(* check controller parameters: (MinOutput > MaxOutput) *)
IF ( MinOutput > MaxOutput ) 
THEN
	ErrorID 												:= ERR_INVALIDPARAM;
	Error													:= TRUE;
	RETURN;
END_IF;

(* check inner and outer window parameters: outer window must be greater than the inner window *)
IF((bIsIPart) AND ( OuterWindow > 0.0 )) 
THEN
	IF (InnerWindow > OuterWindow) 
	THEN
		ErrorId 											:= ERR_INVALIDPARAM;
		Error												:= TRUE;
		RETURN;
	END_IF;
	bIsOuterWnd 											:= TRUE;
END_IF;

(* set internal init flag *)
bIsInitDone													:= TRUE;
Q		 													:= MinOutput;
reset													:= TRUE;
END_METHOD

METHOD PUBLIC synchronize : BOOL  //Return value = TRUE if execution finished
VAR_INPUT 
	IN											:	LREAL;
END_VAR
	MemSyncValue										:= IN;
	
	(* Demand:  SyncValue != Ysum  with  SyncValue = Ysum = YP + YI + YD  =>  YI = SyncValue - Yp - Yd *)
	IF 	( bIsIPart = TRUE ) 
	THEN	(* I-part exists independent from the D-part *)
		(* Normal:  fYI = fYI_1 + fDi * (fE + fE_1) *)
		fYD 											:= fYD_1	:= 0.0;								
		fYI												:= fYI_1	:= MemSyncValue - fYP - fYD;	
		fY												:= MemSyncValue;
	ELSIF ( bIsDPart = TRUE ) 
	THEN	(* no I-part available, only D-part exits *)
		(* Normal:  fYD = fCd * fYD_1 + fDd * (fE - fE_1) *)
		(* fYD := fYD_1 := (fSyncValue - fYP - fYI) / fCd;*)(* 1) pre-calculation for the next cycle; fYI must be zero because there exists no I-part *)
		fYD												:= fYD_1	:= (MemSyncValue - fYP - fYI);		(* 2) fYI must be zero because there exists no I-part *)
		fY												:= MemSyncValue;
	END_IF                              				
	
	Synchronize											:= TRUE;
END_METHOD

END_FUNCTION_BLOCK

// POUs/ControllerTools/PT1Filter
//Low pass filter with a programmable time Tn and factor Kp.
FUNCTION_BLOCK PT1Filter
VAR_INPUT
	Enable													:	BOOL ; 	// FB will be processed as long as enable is TRUE 
	In														:	LREAL := 0.0;	// Actual value
	ResetTrig												:	BOOL ; 	// The function block will be reset with a rising edge 
	Sync													:	BOOL ; 	// Synchronise In to Q - equivalent to Synchronize method
	Kp														:	LREAL := 1.0; 	// Gain
	Tn														:	TIME := T#1S; 	// Integral time 
	Cycletime 												:	TIME := T#10MS;	// cycletime 
END_VAR	            										
VAR_OUTPUT          										
	Q														: LREAL;			// Output
	Error													: BOOL;				// Rising edge of Error informs that an error occurred during the execution of the Function Block 
END_VAR             										
VAR                 	
	Q_old													: LREAL;
END_VAR

(**************************************************************************************
	formula: 
	y(k) = [1-T/T1]	* y(k-1)
			+ T/T1		* v 		* e(k) 
*************************************************************************************)

	Error 													:= Cycletime = T#0MS OR  tn = T#0MS OR Kp = 0.0;
                            								
	IF Enable               								
		AND NOT Error       								
	THEN                    								
		Q 													:=  (1- TIME_TO_LREAL(Cycletime) / TIME_TO_LREAL(Tn))	* Q_old
															 	+ TIME_TO_LREAL(Cycletime) / TIME_TO_LREAL(Tn)	* Kp		* In;
		Q_Old 												:= Q;
	ELSE //Hold
		;
	END_IF

	IF ResetTrig
	THEN
		reset();
	ELSIF Sync
	THEN
		Synchronize(IN);
	END_IF

(************************************************************************************)

METHOD reset : BOOL //Return value = TRUE if execution finished
VAR_INPUT
END_VAR
Q := Q_old 				:= 0.0;
reset				:= TRUE;
END_METHOD

METHOD PUBLIC synchronize : BOOL //Return value = TRUE if execution finished
VAR_INPUT
	IN						:	LREAL;
END_VAR
Q 	:= Q_Old 	 := IN;
Synchronize		:= TRUE;
END_METHOD

END_FUNCTION_BLOCK

// POUs/ControllerTools/signum
//LREAL Signum function
FUNCTION signum : LREAL
VAR_INPUT
	IN		:	LREAL;
END_VAR
VAR
END_VAR

IF IN = 0.0
THEN
	SIGNUM		:= 0.0;
ELSIF IN > 0.0
THEN
	SIGNUM		:= 1.0;
ELSE
	SIGNUM	 	:= -1.0;
END_IF

END_FUNCTION

// POUs/ControllerTools/SlewRateLimitter
//LREAL Slew rate limitter with a timebased change rate
FUNCTION_BLOCK SlewRateLimitter
VAR_INPUT
	IN														: LREAL := 0.0;	 //Actual value
	Sync													: BOOL := FALSE; //Sync signal sets IN to Q	
	Cycletime												: LREAL := 0.001; //cycletime in ms
	Rate													: LREAL := 1.0;	 // changes per second
END_VAR                 									
VAR_OUTPUT              									
	Q														: LREAL := 0.0;   //Output
END_VAR                 									
VAR                     	
	x														: LREAL := 0.0;
END_VAR

//Based on MC_AxUtiSlewRateLimitter_BkPlcMc from TcPlcLibHydraulics , Author WOs
IF Cycletime <= 0.0001 OR Rate <= 0.0 OR Sync
THEN
	Q														:= IN;
ELSE                    									
	x														:= Cycletime * Rate;
	IF ABS(IN) > X OR ABS(Q > In)
	THEN //Start ramping only after In is greater than Rate and as long as Q is greater (if In jumps to zero)
		Q													:= Q + LIMIT(-x , IN - Q , x); 		
	ELSE
		Q													:= In;
	END_IF
END_IF

METHOD PUBLIC synchronize : BOOL //Return value = TRUE if execution finished
VAR_INPUT
	IN														:	LREAL;
END_VAR
Q 															:= IN;
Synchronize 												:= TRUE;
END_METHOD

END_FUNCTION_BLOCK

// POUs/ControllerTools/SlidingAverage
FUNCTION_BLOCK SlidingAverage 
VAR_OUTPUT CONSTANT 
	MIN_BUFFER												:	INT := 1;
	MAX_BUFFER												:	INT := PARAM.SLIDING_AVERAGE_MAX_ENTRYS;
END_VAR
VAR_INPUT
	In														: LREAL := 0.0;			//Actual value 
	ResetTrig												: BOOL := FALSE;		//Reset average buffer
	MaxNoOfValues											: DINT := PARAM.SLIDING_AVERAGE_MAX_ENTRYS;//Buffer limit if value is smaller than MAX_BUFFER
	SampleTime												: TIME := T#0MS;
END_VAR                 									
VAR_OUTPUT              									
	Q														: LREAL := 0.0;			//Average value
	Derivative												: LREAL := 0.0;			//
	ActIdx													: DINT := 1; 			//rotating count of buffer 
	Buffer													: ARRAY [MIN_BUFFER..MAX_BUFFER] OF LREAL;
END_VAR                 									
VAR           
	MinIdx													: DINT := MIN_BUFFER;   
	MaxIdx													: DINT := 0;       									
	Count													: DINT := 0; // limited count 
	pBuffer													: POINTER TO LREAL := 0;
	pIdx													: POINTER TO LREAL := 0;
	IdxOld													: DINT := 1;
	ftotal													: LREAL;
	fttotal													: LREAL;
	tonSampleTimer											: ton;
END_VAR


IF ResetTrig THEN reset(); RETURN; END_IF

pBuffer														:= ADR(Buffer);
MaxIdx														:= LIMIT(MIN_BUFFER, TO_INT(MaxNoOfValues), MAX_BUFFER);

IF(ActIdx>MaxIdx)
THEN
	ActIdx													:= MinIdx;
END_IF                      								
IF(ActIdx<MinIdx)           								
THEN                        								
	ActIdx													:= MaxIdx;
END_IF                      								
                            								
IF(ActIdx>MaxIdx)           								
THEN                        								
	Q														:= IN; (* Puffer-Indices sind unsinnig *)
ELSIF(pBuffer=0)            								
THEN                        								
	Q														:= IN; (* Puffer-Adresse ist unsinnig *)
ELSE            
	tonSampleTimer(IN := SampleTime > T#0MS, PT :=  SampleTime);
	IF NOT tonSampleTimer.IN OR tonSampleTimer.Q    
	THEN   			
		tonSampleTimer(IN := FALSE);	
		
		Count												:= MIN(Count, MaxIdx - MinIdx + 1);
		IdxOld												:= ActIdx - Count;
															
		IF(IdxOld<MinIdx)      								
		THEN                    							
			IdxOld											:= IdxOld + MaxIdx - MinIdx + 1;
		END_IF                  	                        
									                        
		IF(ActIdx=MinIdx)       	                        
		THEN                    	                        
			fttotal											:= 0.0;
		END_IF                  							
															
		IF(Count<1)            								
		THEN                    							
			ftotal := Derivative 							:= 0.0;	(* first cycle *)
		END_IF                  							
															
		pIdx												:= pBuffer + ((ActIdx - MinIdx) * SIZEOF(LREAL));
									                        
		IF(Count = (MaxIdx - MinIdx + 1))                   
		THEN                                                
			Derivative										:= (IN - pIdx^) / DINT_TO_LREAL(Count);
			ftotal											:= ftotal-pIdx^;		(* buffer is filled at least once *)
		END_IF                  							
		pIdx^												:=IN;
		fttotal												:=fttotal + IN;
		ftotal												:=ftotal + IN;
															
		ActIdx												:=ActIdx + 1;
									                        
		IF(ActIdx > MaxIdx)                                 
		THEN                                                
			(* swapping *)                                  
			ftotal											:= fttotal;
			ActIdx											:= MinIdx;
		END_IF                                              
		                                                    
		Count												:= MIN(Count + 1, MaxIdx - MinIdx + 1);
															
		Q													:=ftotal / DINT_TO_LREAL(Count);
	END_IF
END_IF

METHOD PUBLIC reset : BOOL //Return value = TRUE if execution finished
VAR_INPUT
END_VAR
Q															:=0.0;
Derivative													:=0.0;
ActIdx														:=MIN_BUFFER;	(* rotating count *)
Count														:=0;			(* limited count *)
                        									
                        									
IdxOld														:=1;
                        	
ftotal														:=0.0;
fttotal														:=0.0;
MEMSET(ADR(Buffer), 0 , SIZEOF(Buffer));
reset													:= TRUE;
END_METHOD

END_FUNCTION_BLOCK

// POUs/ControllerTools/SlidingAverageExt
//LREAL Sliding average with dynamic allocation of memory according MaxNoofValues 
{attribute 'enable_dynamic_creation'}
FUNCTION_BLOCK SlidingAverageExt 
VAR_INPUT
	In														: LREAL := 0.0;			//Actual value 
	ResetTrig												: BOOL ;		//Reset average buffer
	MaxNoOfValues											: DINT (0..10000) := 0;//Size of buffer (Array size) needs to get assigend in declaration
	SampleTime												: TIME := T#0MS;
END_VAR                 									
VAR_OUTPUT              									
	Q														: LREAL := 0.0;			//Average value
	Derivative												: LREAL := 0.0;			//
	ActIdx													: DINT := 1; 			//rotating count of buffer 
END_VAR                 									
VAR       
	MaxIdx													: DINT := 0;      
	MinIdx													: DINT := 1;        									
	Count													: DINT := 0; // limited count 
	pBuffer													: POINTER TO LREAL := 0;
	pIdx													: POINTER TO LREAL := 0;
	IdxOld													: DINT := 1;
	ftotal													: LREAL;
	fttotal													: LREAL;
	tonSampleTimer											: ton;
END_VAR

(* be sure to have nIdx inside MinIdx..MaxIdx *)
IF pBuffer = 0 AND MaxNoOfValues > 0
THEN //Alocate buffer memory
	pBuffer 												:= __NEW(LREAL,TO_UDINT(MaxNoOfValues)); 	
	IF NOT PARAM.ENABLE_DEBUG_MSG_DYNAMIC_MEM_ALLOCATION
	THEN 
		;
	ELSIF MaxIdx = 0 
	THEN
		AdsLogHint('EngineeringToolbox | FB SlidingAverageExt | An instance allocated %s bytes from the dynamic memory of the ADS router memory pool', TO_STRING(MaxNoOfValues * SIZEOF(LREAL)));	
	ELSE //Allocation of additional memory space
		AdsLogWarn('EngineeringToolbox | FB SlidingAverageExt | Value of "MaxNoOfValues" changed and one instance allocated additional %s bytes from the dynamic memory of the ADS router memory pool', TO_STRING(MaxNoOfValues * SIZEOF(LREAL)));
	END_IF
	MinIdx													:= 1;
	MaxIdx													:= MaxNoOfValues;
ELSIF MaxNoOfValues <> MaxIdx OR MaxNoOfValues = 0
THEN
	reset();
	FB_exit(FALSE);
	RETURN;
END_IF

IF ResetTrig THEN reset(); RETURN; END_IF

IF(ActIdx>MaxIdx)
THEN
	ActIdx													:= MinIdx;
END_IF                      								
IF(ActIdx<MinIdx)           								
THEN                        								
	ActIdx													:= MaxIdx;
END_IF                      								
                            								
IF(ActIdx>MaxIdx)           								
THEN                        								
	Q														:= IN; (* Puffer-Indices sind unsinnig *)
ELSIF(pBuffer=0)            								
THEN                        								
	Q														:= IN; (* Puffer-Adresse ist unsinnig *)
ELSE       
	tonSampleTimer(IN := SampleTime > T#0MS, PT :=  SampleTime);
	IF NOT tonSampleTimer.IN OR tonSampleTimer.Q    
	THEN   			                                        
		tonSampleTimer(IN := FALSE);	                 							
		Count												:= MIN(Count, MaxIdx - MinIdx + 1);
		IdxOld												:= ActIdx - Count;
															
		IF(IdxOld<MinIdx)      								
		THEN                    							
			IdxOld											:= IdxOld + MaxIdx - MinIdx + 1;
		END_IF                  	                        
									                        
		IF(ActIdx=MinIdx)       	                        
		THEN                    	                        
			fttotal											:= 0.0;
		END_IF                  							
															
		IF(Count<1)            								
		THEN                    							
			ftotal := Derivative 							:= 0.0;	(* first cycle *)
		END_IF                  							
															
		pIdx												:= pBuffer + ((ActIdx - MinIdx) * SIZEOF(LREAL));
									                        
		IF(Count = (MaxIdx - MinIdx + 1))                   
		THEN                                                
			Derivative										:= (IN - pIdx^) / DINT_TO_LREAL(Count);
			ftotal											:= ftotal-pIdx^;		(* buffer is filled at least once *)
		END_IF                  							
		pIdx^												:=IN;
		fttotal												:=fttotal + IN;
		ftotal												:=ftotal + IN;
															
		ActIdx												:=ActIdx + 1;
									                        
		IF(ActIdx > MaxIdx)                                 
		THEN                                                
			(* swapping *)                                  
			ftotal											:= fttotal;
			ActIdx											:= MinIdx;
		END_IF                                              
		                                                    
		Count												:= MIN(Count + 1, MaxIdx - MinIdx + 1);
															
		Q													:=ftotal / DINT_TO_LREAL(Count);
	End_If
END_IF

METHOD FB_exit : BOOL 
VAR_INPUT
	bInCopyCode : BOOL; // if TRUE, the exit method is called for exiting an instance that is copied afterwards (online change).
END_VAR
IF NOT bInCopyCode AND pBuffer <> 0
THEN //Release memory in case the PLC stopps
	__DELETE(pBuffer);
	MaxIdx								:= 0;
END_IF
END_METHOD

METHOD PUBLIC reset : BOOL //Return value = TRUE if execution finished
VAR_INPUT
END_VAR
Q															:=0.0;
Derivative													:=0.0;
ActIdx														:=1;			(* rotating count *)
Count														:=0;			(* limited count *)
                        									
                        									
IdxOld														:=1;
                        	
ftotal														:=0.0;
fttotal														:=0.0;


IF pBuffer <> 0
THEN
	MEMSET(pBuffer, 0 , SIZEOF(pBuffer^));
END_IF	

reset														:= TRUE;
END_METHOD

END_FUNCTION_BLOCK

// POUs/Logging/adsLogHint
{attribute 'no_check' := ''}
//Writes a string as a hint message into the TwinCAT AMS Logger and Windows Event Log with an possible argument
//Please see Beckhoff information system "ADSLOGxxxx" for detailed information.
//Intention of this function is to use the handy ADSLOGxxxx with a predefined msgCtrlMask of "ADSLOG_MSGTYPE_STRING OR ADSLOG_MSGTYPE_HINT OR ADSLOG_MSGTYPE_LOG"
FUNCTION adsLogHint : DINT//Write hint message into ADS log windows - Return value will be error code or 0 if OK
VAR_INPUT               											
	MsgFmtStr												:	T_MaxString; ///Message text with %s as placeholder for StrArg
(*	dintArg													:	DINT; //DINT argument for message - to be replaced by %d *) 
	StrArg													:	T_MaxString; //String argument for message - to be replaced by %s
(*	realArg													:	LREAL; //LREAL argument for message - to be replaced by %f *) 
END_VAR
VAR
	msgCtrlMask												:	DWORD; (* 	ADSLOG_MSGTYPE_HINT Meldungstyp ist Hinweis.
																				ADSLOG_MSGTYPE_WARN Meldungstyp ist Warnung.  
																				ADSLOG_MSGTYPE_ERROR Meldungstyp ist Fehler.  
																				ADSLOG_MSGTYPE_LOG Meldung wird in das Logbuch geschrieben.  
																				ADSLOG_MSGTYPE_MSGBOX Meldung wird in einer Messagebox ausgegeben.  
																				ADSLOG_MSGTYPE_RESOURCE Meldung wird aus einer Ressource-Datei geholt. (wird momentan nicht  unterstützt)  
																				ADSLOG_MSGTYPE_STRING 	Meldung ist direkt angegebener String (default).  *)	
END_VAR

(* create fixed message ctrl mask **********************************)
	msgCtrlMask												:= ADSLOG_MSGTYPE_STRING OR ADSLOG_MSGTYPE_HINT OR ADSLOG_MSGTYPE_LOG;

(* write string which includes a floating-number ******************)
(*	AdsLogHint 												:= ADSLOGLREAL(msgCtrlMask, msgFmtStr, realArg); *)
	
(* write string which includes a DINT-number *******************)
(*	AdsLogHint 												:= ADSLOGDINT(msgCtrlMask, msgFmtStr, dintArg); *)

(* write string which includes an other string e.g. 'hallo: %s what's up' ***************)
	adsLogHint 												:= ADSLOGSTR(msgCtrlMask, msgFmtStr,strArg); 

(*****************************************************)

END_FUNCTION

// POUs/Logging/adsLogWarn
{attribute 'no_check' := ''}
//Writes a string as a warining message into the TwinCAT AMS Logger and Windows Event Log with an possible argument
//Please see Beckhoff information system "ADSLOGxxxx" for detailed information.
//Intention of this function is to use the handy ADSLOGxxxx with a predefined msgCtrlMask of "ADSLOG_MSGTYPE_STRING OR ADSLOG_MSGTYPE_WARN OR ADSLOG_MSGTYPE_LOG"
FUNCTION adsLogWarn : DINT//Write warning message into ADS log windows - Return value will be error code or 0 if OK
VAR_INPUT               											
	MsgFmtStr												:	T_MaxString; //Message text with %s as placeholder for StrArg
(*	dintArg													:	DINT; //DINT argument for message - to be replaced by %d *) 
	StrArg													:	T_MaxString; //String argument for message - to be replaced by %s
(*	realArg													:	LREAL; //LREAL argument for message - to be replaced by %f *) 
END_VAR
VAR
	msgCtrlMask												:	DWORD; (* 	ADSLOG_MSGTYPE_HINT Meldungstyp ist Hinweis.
																				ADSLOG_MSGTYPE_WARN Meldungstyp ist Warnung.  
																				ADSLOG_MSGTYPE_ERROR Meldungstyp ist Fehler.  
																				ADSLOG_MSGTYPE_LOG Meldung wird in das Logbuch geschrieben.  
																				ADSLOG_MSGTYPE_MSGBOX Meldung wird in einer Messagebox ausgegeben.  
																				ADSLOG_MSGTYPE_RESOURCE Meldung wird aus einer Ressource-Datei geholt. (wird momentan nicht  unterstützt)  
																				ADSLOG_MSGTYPE_STRING 	Meldung ist direkt angegebener String (default).  *)	
END_VAR

(* create fixed message ctrl mask **********************************)
	msgCtrlMask												:= ADSLOG_MSGTYPE_STRING OR ADSLOG_MSGTYPE_WARN OR ADSLOG_MSGTYPE_LOG;

(* write string which includes a floating-number ******************)
(*	AdsLogWarn 												:= ADSLOGLREAL(msgCtrlMask, msgFmtStr, realArg); *)
	
(* write string which includes a DINT-number *******************)
(*	AdsLogWarn 												:= ADSLOGDINT(msgCtrlMask, msgFmtStr, dintArg); *)

(* write string which includes an other string e.g. 'hallo: %s what's up' ***************)
	adsLogWarn 												:= ADSLOGSTR(msgCtrlMask, msgFmtStr,strArg); 

(*****************************************************)

END_FUNCTION

// POUs/ControllerTools/ThreePointController
//Three point controller with lreal output
//The On-Values must be greater then the Off-Values. The difference is equivalent to the hysteresis-value
FUNCTION_BLOCK ThreePointController 
VAR_INPUT
	Enable													: BOOL := TRUE;		//Enable controller	
	SetValue												: LREAL := 0.0;		//Setpoint value
	ActValue												: LREAL := 0.0;		//Actual value
	
	Sync													: BOOL := FALSE; 	//Synchronization flag for bumpless initialisation		
	SyncValue												: LREAL := 0.0; 	//Syncronization value for bumpless init.			
	MinOutput												: LREAL := 0.0; 	//Controller minimum analog output			
	MaxOutput												: LREAL := 100.0;	//Controller maximum analog output (Limitation is switched off at 0.0) 			

	FeedPlus												: BOOL := TRUE;		//Release for controller plus 
	FeedMinus												: BOOL := TRUE;		//Release for controller minus 
	                                						
	ManualOn												: BOOL := FALSE;	//Manual mode on - set analog output to ManualValue
	ManualValue												: LREAL	:= 0.0;		//Analog output in manual mode
	ManualPlus												: BOOL := FALSE;	//Manual control of digital plus output	
	ManualMinus												: BOOL := FALSE;	//Manual control of digital minus output	
                                    						
	Stepwide												: LREAL := 1.0; 	//Stepwidth analog output
	Breaktime												: TIME := T#500MS; 	//Breaktime after a change of output
	DriveTime												: TIME := T#500MS; 	//Drivetime for digital outputs  
	                                					
	PlusOn													: LREAL := 5.0;		//Derivate hysteresis to increase the controller output (need to be greater than PlusOff , Plus or Minus pair need to be less the zero)  
	PlusOff													: LREAL := 3.0;		//Derivate hysteresis to switch off the controller output (need to be smaller than PlusOn , Plus or Minus pair need to be less the zero  
	MinusOff												: LREAL := -3.0;	//Derivate hysteresis to switch the controller output (need to be greater smaller than MinusOn , Plus or Minus pair need to be less the zero) 
	MinusOn													: LREAL := -5.0;	//Derivate hysteresis to decrease the controller output (need to be greater than MinusOff , Plus or Minus pair need to be less the zero)
END_VAR                             						
VAR_OUTPUT	   
	Q														: LREAL; 			//Analog controller output
	Q_Plus													: BOOL;				//Digital controller output
	Q_Minus													: BOOL;				//Digital controller output
	Deviation												: LREAL;			//deviation between actual value and setpoint (Deviation = SetValue - ActValue)
	DeadZone												: LREAL;			//Active dead zone based on PlusOn/Off and MinusOn/Off values
	BreakTimeRunning										: BOOL;				//Controller is on hold - Break time running 
	DriveTimeRunning										: BOOL;				//Controller is active 
	Error													: BOOL;             //Error occured       						
END_VAR                             						
VAR 
//local variables *********************************************************          
	state													: INT;     
	MemPlus													: BOOL;
	MemMinus												: BOOL;
	Cooling													: BOOL;      

//Trigger ****************************************************************           						
	rtSync													: r_trig;	
	
//timer ******************************************************************
	tonBreakTime											:	ton;
	tonDriveTime											:	ton;

	
END_VAR

(* 3 point bang-bang controller 	 							*)
(****************************************************************)

IF ABS(MinusOn) <= ABS(MinusOff) //On offset must be greater then off
	OR ABS(PlusOn) <= ABS(PlusOff) //Off offsetr must be smallet then on
	OR NOT(MinusOn > 0.0 XOR PlusOn > 0.0)//Only one offset needs to be greater then 0.0
	OR NOT(PlusOff > 0.0 XOR MinusOff > 0.0)//Only one offset needs to be greater then 0.0
	OR MinOutput > MaxOutput AND MaxOutput <> 0.0
THEN
	reset();
	Error													:= Enable;
ELSE                                            			
	rtSync(CLK := Sync);                        			
	IF rtSync.Q                                 			
	THEN                                        			
		Synchronize(SyncValue); 
	END_IF                                      			
	                                            			
	Error													:= FALSE;
	DeadZone												:= ABS(PlusOff) + ABS(MinusOff);
	Deviation												:= SetValue - ActValue; 
	Cooling													:= PlusOn < 0.0 AND MinusOn > 0.0;
		  
	//Control sequecne                                      			
	CASE state OF                               			
	0:                                          			
		//Check wheter controller needs to start 
		IF ManualON                             			
		THEN                                    			
			MemMinus := MemPlus								:= FALSE;
			Q												:= ManualValue;
		ELSIF NOT Enable                        			
		THEN                                    			
			reset();
		ELSIF(Q < MaxOutput OR MaxOutput = 0.0)       
			AND FeedPlus    			
			AND(                                			
			Deviation > PlusOn AND NOT Cooling     			
			OR  Deviation < PlusOn AND Cooling)     			
		THEN // greatest Plusitive deviatoin      			
			MemPlus											:= TRUE;
			MemMinus										:= FALSE;
		ELSIF(Q > MinOutput OR MaxOutput = 0.0)    
			AND FeedMinus      			
			AND(                                			
			Deviation < MinusOn AND NOT Cooling      	
			OR Deviation > MinusOn AND Cooling)      			
		THEN // greatest Minusative deviation     			
			MemMinus										:= TRUE;
			MemPlus											:= FALSE;
			
		ELSE
			MemPlus											:= MemPlus AND ABS(Deviation) >= ABS(PlusOff) ;
			MemMinus										:= MemMinus AND ABS(Deviation) >= ABS(MinusOff);
		END_IF              			
		                       
		//Continue to run controller up or down as long as memory is still active                  			
		IF MemMinus	                            			
		THEN                                    			
			Q												:= MAX(Q - Stepwide, MinOutput);
			state											:= 1;
		ELSIF MemPlus                            			
		THEN                                    			
			Q												:= MIN(Q + Stepwide, MaxOutput);
			state											:= 1;
		ELSE                                    			
			Q												:= LIMIT(MinOutput, Q, MaxOutput);
		END_IF		
			
	1: //start drive time 
		tonDriveTime(IN := FALSE); tonBreakTime(IN := FALSE);
		IF DriveTime > T#0MS
		THEN
			tonDriveTime(IN := TRUE, PT := DriveTime);
			state											:= 2;
		ELSIF BreakTime > T#0MS
		THEN
			tonBreakTime(IN := TRUE, PT := BreakTime);	
			state											:= 3;	
		ELSE
			state											:= 0;			
		END_IF
				                    			
	2:  //run drive time                                       			
		tonDriveTime();
		IF ManualOn
		THEN
           state											:= 0;    			
		ELSIF tonDriveTime.Q                			
		THEN
			IF BreakTime > T#0MS
			THEN
				tonBreakTime(IN := TRUE, PT := BreakTime);
				state										:= 3;
			ELSE
				state										:= 0;				
			END_IF				             	
		END_IF     
                    
	3: //run break time 
		tonBreakTime();
		IF ManualOn OR tonBreakTime.Q  
		THEN
           state											:= 0;    			
		END_IF	
	END_CASE                                    			
	
	//status
	DriveTimeRunning										:= state = 2;
	BreakTimeRunning										:= state = 3;
                                            			                      			                                                		
	//setting ouputs
	Q_Minus 												:= FeedMinus AND Enable
																AND(
																MemMinus AND DriveTimeRunning 
																OR ManualOn AND ManualMinus) ;
										
	Q_Plus				 									:= FeedPlus AND Enable
																AND(
																MemPlus AND DriveTimeRunning
																OR ManualOn AND ManualPlus) ;
																						
END_IF

METHOD PUBLIC reset : booL //Return value = TRUE if execution finished
VAR_INPUT
END_VAR
Q												:= MinOutput;
MemMinus := MemPlus								:= FALSE;
state											:= 0;

Q_Plus											:= FALSE;
Q_Minus											:= FALSE;
Error											:= FALSE;
Deviation										:= 0.0;
DeadZone										:= 0.0;
BreakTimeRunning								:= FALSE;
DrivetimeRunning								:= FALSE;

reset										:= TRUE;
END_METHOD

METHOD PUBLIC synchronize : BOOL //Return value = TRUE if execution finished
VAR_INPUT
	IN											:	LREAL;
END_VAR
Q								:= LIMIT(MinOutput,IN,MaxOutput);
Synchronize						:= TRUE;
END_METHOD

END_FUNCTION_BLOCK

// POUs/DataBuffer/FiFo/Fifo
//Fifo base control template with external memory based of FifoBase
FUNCTION_BLOCK Fifo EXTENDS FifoBase
VAR_INPUT
END_VAR
VAR_OUTPUT
END_VAR
VAR
END_VAR

;

//Clear out one entry from the Fifo buffer
METHOD PUBLIC clear : BOOL //TRUE if method was successful
VAR_INPUT
	EntryNo													:	UDINT;
	pMemory													: 	POINTER TO BYTE := 0;
	SizeOfMemory											: 	UDINT := 0;
END_VAR             										
VAR                 										
END_VAR
Clear := SUPER^._Clear(EntryNo,pMemory,SizeOfMemory);
END_METHOD

//Clear out defined data set from the Fifo buffer
METHOD PUBLIC clearByDataSet : BOOL //TRUE if method was successful
VAR_INPUT
	pData													: 	POINTER TO BYTE := 0;
	SizeOfData												: 	UDINT := 0;										
	pMemory													: 	POINTER TO BYTE := 0;
	SizeOfMemory											: 	UDINT := 0;
END_VAR             										
VAR         
	i														:	DINT;        										
END_VAR
ClearByDataSet := SUPER^._ClearByDataSet(pData,SizeOfEntry,pMemory,SizeOfMemory);
END_METHOD

METHOD PUBLIC dequeue : BOOL //TRUE if method was successful
VAR_INPUT
	pData													: 	POINTER TO BYTE := 0;
	SizeOfData												: 	UDINT := 0;
	pMemory													: 	POINTER TO BYTE := 0;
	SizeOfMemory											: 	UDINT := 0;
END_VAR
Dequeue := SUPER^._Dequeue(pData,SizeOfEntry,pMemory,SizeOfMemory);
END_METHOD

METHOD PUBLIC enqueue : BOOL //TRUE if method was successful
VAR_INPUT
	pData													: 	POINTER TO BYTE := 0;
	SizeOfData												: 	UDINT := 0;
	pMemory													: 	POINTER TO BYTE := 0;
	SizeOfMemory											: 	UDINT := 0;
END_VAR
Enqueue := SUPER^._Enqueue(pData,SizeOfData,pMemory,SizeOfMemory);
END_METHOD

//Check wheter a value already exist
METHOD PUBLIC isEnqueued : uDINT //data exist in Fifo if reurn value <> 0, returns index of entry in buffer 
VAR_INPUT
	pData													: 	POINTER TO BYTE := 0;
	SizeOfData												: 	UDINT := 0;
	pMemory													: 	POINTER TO BYTE := 0;
	SizeOfMemory											: 	UDINT := 0;
END_VAR	
VAR
	i 														: 	DINT;
END_VAR
IsEnqueued := SUPER^._IsEnqueued(pData,SizeOfEntry,pMemory,SizeOfMemory);
END_METHOD

//Check wheter a value will be the next output of the buffer
METHOD PUBLIC isNextEntry : BOOL //Inputs value is the next output 
VAR_INPUT
	pData													: 	POINTER TO BYTE := 0;
	SizeOfData												: 	UDINT := 0;
	pMemory													: 	POINTER TO BYTE := 0;
	SizeOfMemory											: 	UDINT := 0;
END_VAR
VAR
END_VAR
IsNextEntry := SUPER^._IsNextEntry(pData,SizeOfEntry,pMemory,SizeOfMemory);
END_METHOD

METHOD PUBLIC readEntry : BOOL //TRUE if method was successful
VAR_INPUT
	idx														:	UDINT;
	pData													: 	POINTER TO BYTE := 0;
	SizeOfData												: 	UDINT := 0;
	pMemory													: 	POINTER TO BYTE := 0;
	SizeOfMemory											: 	UDINT := 0;
END_VAR
ReadEntry := SUPER^._ReadEntry(idx,pData,SizeOfEntry,pMemory,SizeOfMemory);
END_METHOD

//Reset complete Fifo
METHOD PUBLIC reset : BOOL //TRUE if method is finnished
VAR_INPUT
	pMemory													: 	POINTER TO BYTE := 0;
	SizeOfMemory											: 	UDINT := 0;
END_VAR
reset := SUPER^._reset(pMemory,SizeOfMemory);
END_METHOD

END_FUNCTION_BLOCK

// POUs/DataBuffer/FiFo/FiFoBase
//Fifo basic control template with external memory 
FUNCTION_BLOCK FiFoBase
VAR_INPUT
	Overwrite												:	BOOL := FALSE; //Return value TRUE = overwrite oldest entry 
END_VAR
VAR_OUTPUT
	Count													:	UDINT := 0; //Number of entrys	
	Full													:	BOOL := FALSE; //Fifo is full
	Empty													:	BOOL := TRUE;  //Fifo is empty
END_VAR
VAR
	Interlock												:	BOOL; //Multitask interlock
	MaxEntrys												:	UDINT := 0; //Maximum number of entrys based on size of data and size of memory
	SizeOfEntry												:	UDINT := 0;
END_VAR

;

//Clear out one entry from the Fifo buffer
METHOD PROTECTED _clear : BOOL //TRUE if method was successful
VAR_INPUT
	EntryNo													:	UDINT;
	pMemory													: 	POINTER TO BYTE := 0;
	SizeOfMemory											: 	UDINT := 0;
END_VAR             										
VAR                 										
END_VAR
IF EntryNo = 0
	OR pMemory = 0
	OR SizeOfMemory = 0
THEN
	_Clear													:= FALSE;
	RETURN;
ELSIF TestAndSet(Interlock)
THEN	
	IF Empty OR EntryNo > Count
	THEN
		_Clear												:=TRUE;
	ELSE	                        						
		MaxEntrys 											:= SizeOfMemory / SizeOfEntry;	
		
		//shift datasets
		MEMMOVE(pMemory + ((EntryNo - 1) * SizeOfEntry) , pMemory + (EntryNo * SizeOfEntry)  , (Count - EntryNo) * SizeOfEntry);
		
		//delete last shifted dataset 
		MEMSET(pMemory + ((Count - 1) * SizeOfEntry),0, SizeOfEntry);

		Count 												:= MAX(0,Count - 1);
		Full 												:= FALSE;
		Empty 												:= Count = 0;
		_Clear												:= TRUE;	
	END_IF
	Interlock												:= FALSE;
ELSE
	_Clear													:= FALSE;
END_IF
END_METHOD

//Clears out defined data set from the Fifo buffer
METHOD PROTECTED _clearByDataSet : BOOL //TRUE if method was successful
VAR_INPUT
	pData													: 	POINTER TO BYTE := 0;
	SizeOfData												: 	UDINT := 0;										
	pMemory													: 	POINTER TO BYTE := 0;
	SizeOfMemory											: 	UDINT := 0;
END_VAR             										
VAR         
	i														:	UDINT;        										
END_VAR
IF 	pData = 0
	OR SizeOfData = 0
	OR pMemory = 0
	OR SizeOfMemory = 0
	OR Empty
THEN
	_ClearByDataSet											:= FALSE;
	RETURN;
ELSIF TestAndSet(Interlock)
THEN
	_ClearByDataSet											:= FALSE;
	MaxEntrys 												:= SizeOfMemory / SizeOfData;	
	FOR i := Count TO 1 BY -1
	DO
		
		IF MEMCMP(pData,pMemory + ((i - 1) * SizeOfData), SizeOfData) = 0
		THEN
			IF TO_UDINT(i) >= MaxEntrys
			THEN //Just delete the entry at the end of the list
				MEMSET(pMemory + ((i - 1) * SizeOfData),0, SizeOfData);
				Count 										:= MAX(0,Count - 1);
			ELSE //Copy the other entrys over the found one and delte the left entry from the list
				MEMMOVE(pMemory + ((i - 1) * SizeOfData),pMemory + (i * SizeOfData) , MIN(Count - i, MaxEntrys - 1) * SizeOfData);
				MEMSET(pMemory + ((Count - 1 )* SizeOfData),0, SizeOfData);
				Count 										:= MAX(0,Count - 1);
			END_IF		
			_ClearByDataSet									:= TRUE;
			Full 											:= FALSE;
			Empty 											:= Count = 0;		
			IF Empty 
			THEN
				EXIT;
			END_IF
		END_IF
	END_FOR
	Interlock												:= FALSE;
END_IF
END_METHOD

METHOD PROTECTED _dequeue : BOOL //TRUE if method was successful
VAR_INPUT
	pData													: 	POINTER TO BYTE := 0; //pointer to destination of data
	SizeOfData												: 	UDINT := 0; //Size of destination data
	pMemory													: 	POINTER TO BYTE := 0;
	SizeOfMemory											: 	UDINT := 0;
END_VAR
IF 	pData = 0
	OR SizeOfData = 0
	OR pMemory = 0
	OR SizeOfMemory = 0
	OR Empty
THEN
	_Dequeue												:= FALSE;
	RETURN;
ELSIF TestAndSet(Interlock)
THEN	
	(* copy dataset *)
	MEMMOVE(pData,pMemory + (MAX(0, (Count - 1)) * SizeOfData),SizeOfData);
	
	(* delete dataset *)
	MEMSET(pMemory + (MAX(0,(Count - 1)) * SizeOfData) ,0 ,SizeOfData);
	Count 													:= MAX(0,Count - 1);
	Full 													:= FALSE;
	Empty 													:= Count = 0;
	_Dequeue												:= TRUE;
	Interlock												:= FALSE;
ELSE
	_Dequeue												:= FALSE;
END_IF
END_METHOD

METHOD PROTECTED _enqueue : BOOL //TRUE if method was successful
VAR_INPUT
	pData													: 	POINTER TO BYTE := 0;
	SizeOfData												: 	UDINT := 0;
	pMemory													: 	POINTER TO BYTE := 0;
	SizeOfMemory											: 	UDINT := 0;
END_VAR
IF pData = 0
	OR SizeOfData = 0
	OR pMemory = 0
	OR SizeOfMemory = 0
	OR Full AND NOT Overwrite
THEN
	_Enqueue												:= FALSE;
	RETURN;
ELSIF TestAndSet(Interlock)
THEN	
	_Enqueue												:= TRUE;
		
	(* maximum count *)
	MaxEntrys 												:= SizeOfMemory / SizeOfData;
	SizeOfEntry												:= SizeOfData;

	(* copy datasets *)
	MEMMOVE(pMemory + SizeOfData, pMemory, SEL(Full AND Overwrite,Count * SizeOfData , (Count - 1) * SizeOfData));
	
	(* copy datasets at the beginning *)
	MEMCPY(pMemory,pData,SizeOfData);
	Count													:= MIN(Count + 1, MaxEntrys);
	Empty 													:= FALSE;
	Full 													:= Count >= MaxEntrys;
	Interlock												:= FALSE;
ELSE
	_Enqueue												:= FALSE;
END_IF
END_METHOD

//Check wheter a value already exist
METHOD PROTECTED _isEnqueued : UDINT //data exist in Fifo if reurn value <> 0, returns index of entry in buffer 
VAR_INPUT
	pData													: 	POINTER TO BYTE := 0;
	SizeOfData												: 	UDINT := 0;
	pMemory													: 	POINTER TO BYTE := 0;
	SizeOfMemory											: 	UDINT := 0;
END_VAR	
VAR
	i 														: 	UDINT;
END_VAR
IF 	pData = 0
	OR SizeOfData = 0
	OR pMemory = 0
	OR SizeOfMemory = 0
	OR Empty
THEN
	_IsEnqueued												:= 0;
	RETURN;
ELSIF TestAndSet(Interlock)
THEN	
	_IsEnqueued												:= 0;
	MaxEntrys 												:= SizeOfMemory / SizeOfData;
	FOR i := 1 TO Count
	DO
		IF MEMCMP(pData,pMemory + ((i - 1) * SizeOfData), SizeOfData) = 0
		THEN
			_isEnqueued										:= i;
			EXIT;
		END_IF
	END_FOR
	Interlock												:= FALSE;
END_IF
END_METHOD

//Check wheter a value will be the next output of the buffer
METHOD PROTECTED _isNextEntry : BOOL //Inputs value is the next output 
VAR_INPUT
	pData													: 	POINTER TO BYTE := 0;
	SizeOfData												: 	UDINT := 0;
	pMemory													: 	POINTER TO BYTE := 0;
	SizeOfMemory											: 	UDINT := 0;
END_VAR
VAR
END_VAR
_IsNextEntry 	:= 0 = MEMCMP(pData,pMemory +(TO_UDINT(Count -1) * SizeOfData), SizeOfData) and NOT Empty;
END_METHOD

METHOD PROTECTED _readEntry : BOOL //TRUE if method was successful
VAR_INPUT
	idx														:	UDINT;
	pData													: 	POINTER TO BYTE := 0;
	SizeOfData												: 	UDINT := 0;
	pMemory													: 	POINTER TO BYTE := 0;
	SizeOfMemory											: 	UDINT := 0;
END_VAR
IF 	pData = 0
	OR SizeOfData = 0
	OR pMemory = 0
	OR SizeOfMemory = 0
	OR Empty
THEN
	_ReadEntry												:= FALSE;
	RETURN;
ELSIF TestAndSet(Interlock)
THEN	
	MaxEntrys 												:= SizeOfMemory / SizeOfData;
	IF idx < 1 OR idx > MIN(Count,MaxEntrys)
	THEN
		_ReadEntry											:= FALSE;
	ELSE
		MEMCPY(pData,pMemory + ((idx - 1) * SizeOfData), SizeOfData);
		_ReadEntry											:= TRUE;					
	END_IF
	Interlock												:= FALSE;
END_IF
END_METHOD

//Reset complete Fifo
METHOD PROTECTED _reset : BOOL //TRUE if method is finnished
VAR_INPUT
	pMemory													: 	POINTER TO BYTE := 0;
	SizeOfMemory											: 	UDINT := 0;
END_VAR
IF pMemory = 0
	OR SizeOfMemory = 0
THEN
	_reset													:= FALSE;
	RETURN;
ELSIF TestAndSet(Interlock)
THEN
	(* delete *)
	MEMSET(pMemory,0,SizeOfMemory);
	Empty 													:= TRUE;
	Full 													:= FALSE;
	Count 													:= 0;
	_reset													:= TRUE;
	Interlock												:= FALSE;
ELSE
	_reset													:= TRUE;
END_IF
END_METHOD

END_FUNCTION_BLOCK

// POUs/DataBuffer/FiFo/FiFoExt
//FifoBase extended with dynamical memory allocation
 {attribute 'enable_dynamic_creation'}
FUNCTION_BLOCK FiFoExt EXTENDS FifoBase
VAR_OUTPUT CONSTANT
END_VAR   
VAR_INPUT
	MaxNoOfEntrys											: 	UDINT := 10;	//0 = dynamically allocation / <> 0 = pre allcoation of memory based on size of first entry (n * data size) 
END_VAR
VAR_OUTPUT
	pMemory													: 	POINTER TO BYTE := 0; //Pointer to memory	
	SizeOfMemory											: 	UDINT := 0; //According MaxNoOfEntrys and SizeOfData of first entry
END_VAR
VAR
	MemSizeAllocatedMemory									:	UDINT := 0; //Allocated memory 
	MemSizeOfData											:	UDINT;
	MemMaxNoOfEntrys										:	UDINT;
	ExtInterlock											:	BOOL;
END_VAR

;

METHOD PROTECTED FINAL allocate : BOOL
VAR_IN_OUT
	SizeOfData												:	UDINT;
END_VAR
VAR
	pDummy													:	POINTER TO BYTE;	
End_Var
IF pMemory = 0
THEN
	IF SizeOfData = 0 OR MaxNoOfEntrys = 0
	THEN
		Allocate											:= FALSE;	
	ELSE
		MemSizeOfData										:= SizeOfData;
		MemMaxNoOfEntrys									:= MaxNoOfEntrys;
		SizeOfMemory										:= MemSizeOfData * MemMaxNoOfEntrys;
		MemSizeAllocatedMemory								:= SizeOfMemory;
		pMemory												:= __NEW(BYTE,SizeOfMemory );
		
		IF PARAM.ENABLE_DEBUG_MSG_DYNAMIC_MEM_ALLOCATION
		THEN
			AdsLogHint('EngineeringToolbox | FB FifoExt | An instance allocated %s bytes from the dynamic memory of the ADS router memory pool', TO_STRING(SizeOfMemory));
		END_IF
	END_IF

ELSIF SizeOfData = MemSizeOfData AND MaxNoOfEntrys = MemMaxNoOfEntrys
THEN
	Allocate												:= TRUE;
	
ELSIF SizeOfData > MemSizeOfData OR MaxNoOfEntrys > MemMaxNoOfEntrys
THEN //Since increased, allocate new memory
	MemSizeAllocatedMemory									:= SizeOfData * MaxNoOfEntrys;
	pDummy													:= __NEW(BYTE, MemSizeAllocatedMemory); 
	
	 //Size of data still the same, copy old data to reuse
	IF MemSizeOfData = SizeOfData AND Count > 0
	THEN
		MEMCPY(pDummy,pMemory, SizeOfMemory);
	END_IF
	
	//Copy new settings to local variales
	MemSizeOfData											:= SizeOfData;
	MemMaxNoOfEntrys										:= MaxNoOfEntrys;	
	SizeOfMemory 											:= MemSizeAllocatedMemory;

	__DELETE(pMemory);  //Delete reference to old memory
	pMemory													:= pDummy; //Take over new pointer to new memory
	
	IF PARAM.ENABLE_DEBUG_MSG_DYNAMIC_MEM_ALLOCATION
	THEN
		AdsLogWarn('EngineeringToolbox | FB FifoExt | Value of "MaxNoOfEntrys" or data size increased and one instance allocated additional %s bytes from the dynamic memory of the ADS router memory pool', TO_STRING(SizeOfMemory));
	END_IF
	
	Allocate												:= TRUE;
	
ELSE //Size decreased
	IF MemSizeOfData <> SizeOfData AND Count > 0
	THEN //Size of data changed, erease memory 
		MEMSET(pMemory,0, MemSizeAllocatedMemory);
	ELSE //Size of data the same, keep current data
		;
	END_IF
	
	//Copy new settings to local variales
	MemSizeOfData											:= SizeOfData;
	MemMaxNoOfEntrys										:= MaxNoOfEntrys;
	SizeOfMemory											:= MemSizeOfData * MemMaxNoOfEntrys;
	Allocate												:= TRUE;
END_IF
END_METHOD

//Clear out one entry from the Fifo buffer
METHOD PUBLIC clear : BOOL //TRUE if method was successful
VAR_INPUT
	EntryNo													:	UDINT;
END_VAR             										
VAR                 										
END_VAR
Clear := SUPER^._Clear(EntryNo,This^.pMemory,This^.SizeOfMemory);
END_METHOD

//Clear out defined data set from the Fifo buffer
METHOD PUBLIC clearByDataSet : BOOL //TRUE if method was successful
VAR_INPUT
	pData													: 	POINTER TO BYTE := 0;				
END_VAR             										
VAR                 										
END_VAR
ClearByDataSet := SUPER^._ClearByDataSet(pData,SizeOfEntry,This^.pMemory,This^.SizeOfMemory);
END_METHOD

METHOD PUBLIC dequeue : BOOL //TRUE if method was successful
VAR_INPUT
	pData													:	POINTER TO BYTE;	
END_VAR
VAR
END_VAR
Dequeue := SUPER^._Dequeue(pData,SizeOfEntry,This^.pMemory,This^.SizeOfMemory);
END_METHOD

METHOD PUBLIC enqueue : BOOL //TRUE if method was successful
VAR_INPUT
	pData													:	POINTER TO BYTE;
	SizeOfData												:	UDINT;
END_VAR
VAR
	CopySize												:	UDINT;
	pDummy													:	POINTER TO BYTE;
END_VAR
IF TestAndSet(ExtInterlock) 
THEN	
	if Allocate(SizeOfData)
	then
		Enqueue 											:= SUPER^._Enqueue(pData,SizeOfData,THIS^.pMemory,THIS^.SizeOfMemory);
		ExtInterlock										:= FALSE;
	else
		Enqueue												:= FALSE;
	END_IF	
ELSE
	Enqueue													:= FALSE;
END_IF
END_METHOD

METHOD FB_exit : BOOL
VAR_INPUT
	bInCopyCode : BOOL; // if TRUE, the exit method is called for exiting an instance that is copied afterwards (online change).
END_VAR
IF NOT bInCopyCode AND pMemory <> 0
THEN //Release memory in case the PLC stopps
	__DELETE(pMemory);
	Full													:= FALSE;
	Empty													:= TRUE;
	Count													:= 0;
	SizeOfMemory											:= 0;
	MemSizeOfData											:= 0;
	MemSizeAllocatedMemory									:= 0;
	MemMaxNoOfEntrys										:= MaxNoOfEntrys;
END_IF
END_METHOD

//Check wheter a value already exist
METHOD PUBLIC isEnqueued : UDINT //pData entry exist in Fifo at idx as return value 
VAR_INPUT
	pData													: 	POINTER TO BYTE := 0;
END_VAR
IsEnqueued := SUPER^._IsEnqueued(pData,SizeOfEntry,This^.pMemory,This^.SizeOfMemory);
END_METHOD

//Check wheter a value will be the next output of the buffer
METHOD PUBLIC isNextEntry : BOOL //Inputs value is the next output 
VAR_INPUT
	pData													: 	POINTER TO BYTE := 0;
END_VAR
VAR
END_VAR
IsNextEntry := SUPER^._IsNextEntry(pData,SizeOfEntry,This^.pMemory,This^.SizeOfMemory);
END_METHOD

METHOD PUBLIC readEntry : BOOL //TRUE if method was successful
VAR_INPUT
	idx														:	UDINT;
	pData													: 	POINTER TO BYTE := 0;
END_VAR
ReadEntry := SUPER^._ReadEntry(idx,pData,SizeOfEntry,This^.pMemory,This^.SizeOfMemory);
END_METHOD

//Reset complete Fifo
METHOD PUBLIC reset : BOOL //TRUE if method is finnished
VAR_INPUT
END_VAR
reset				:= SUPER^._reset(This^.pMemory,This^.SizeOfMemory);
END_METHOD

END_FUNCTION_BLOCK

// POUs/DataBuffer/FiFo/FiFoLRealSimple
//Fifo with a internal Lreal array for a simple num list implementation
FUNCTION_BLOCK FiFoLRealSimple EXTENDS FifoBase
VAR_OUTPUT CONSTANT
	MIN_BUFFER												:	DINT := 1; //Fifo buffer start index 
	MAX_BUFFER												:	DINT := PARAM.FIFO_LREAL_SIMPEL_MAX_BUFFER; //Fifo buffer end index - see library parameter to customize parameter
END_VAR   
VAR_INPUT
END_VAR
VAR_OUTPUT
	Buffer													:	ARRAY[MIN_BUFFER..MAX_BUFFER] OF LREAL; //Lreal Fifo buffer 
END_VAR
VAR
END_VAR

;

 //Clear out one entry from the Fifo buffer
METHOD PUBLIC clear : BOOL //TRUE if method was successful
VAR_INPUT
	EntryNo													:	UDINT;
END_VAR             										
VAR                 										
END_VAR
Clear := super^._Clear(EntryNo,ADR(Buffer),SIZEOF(Buffer));
END_METHOD

//Clear out defined data set from the Fifo buffer
METHOD PUBLIC clearByDataSet : BOOL //TRUE if method was successful
VAR_INPUT
	Value													:	LREAL;
END_VAR             										
VAR                 										
END_VAR
ClearByDataSet := super^._ClearByDataSet(ADR(Value),SIZEOF(Value),ADR(Buffer),SIZEOF(Buffer));
END_METHOD

METHOD PUBLIC dequeue : BOOL //TRUE if method was successful
VAR_IN_OUT
	Value													:	LREAL;	
END_VAR
VAR
END_VAR
Dequeue := SUPER^._Dequeue(ADR(Value),SIZEOF(Value),ADR(Buffer),SIZEOF(Buffer));
END_METHOD

METHOD PUBLIC enqueue : BOOL //TRUE if method was successful
VAR_INPUT
	Value													:	LREAL;
END_VAR
Enqueue := SUPER^._Enqueue(ADR(Value),SIZEOF(Value),ADR(Buffer),SIZEOF(Buffer));
END_METHOD

//Check wheter a value already exist
METHOD PUBLIC isEnqueued : uDINT //In Value exist in Fifo at idx as return value  
VAR_INPUT
	Value													:	LREAL;
END_VAR
IsEnqueued := SUPER^._IsEnqueued(ADR(Value),SIZEOF(Value),ADR(Buffer),SIZEOF(Buffer));
END_METHOD

//Check wheter a value will be the next output of the buffer
METHOD PUBLIC isNextEntry : BOOL //Inputs value is the next output 
VAR_INPUT
	Value													: LREAL;
END_VAR
VAR
END_VAR
IsNextEntry := SUPER^._IsNextEntry(ADR(Value),SIZEOF(Value),ADR(Buffer),SIZEOF(Buffer));
END_METHOD

METHOD PUBLIC readEntry : BOOL //TRUE if method was successful
VAR_INPUT
	idx														:	uDINT;
END_VAR
VAR_IN_OUT
	value													: LREAL;	
END_VAR
ReadEntry := SUPER^._ReadEntry(idx,ADR(Value),SIZEOF(Value),ADR(Buffer),SIZEOF(Buffer));
END_METHOD

//Reset complete Fifo
METHOD PUBLIC reset : BOOL //TRUE if method is finnished
VAR_INPUT
END_VAR
reset := SUPER^._reset(ADR(Buffer),SIZEOF(Buffer));
END_METHOD

END_FUNCTION_BLOCK

// POUs/DataBuffer/LiFo/LiFo
//LiFo base control template with external memory based of LifoBase
FUNCTION_BLOCK LiFo EXTENDS LifoBase
VAR_INPUT
END_VAR
VAR_OUTPUT
END_VAR
VAR
END_VAR

;

METHOD PUBLIC dequeue : BOOL //TRUE if method was successful
VAR_INPUT
	pData													: 	POINTER TO BYTE := 0;
	SizeOfData												: 	UDINT := 0;
	pMemory													: 	POINTER TO BYTE := 0;
	SizeOfMemory											: 	UDINT := 0;
END_VAR
Dequeue := SUPER^._Dequeue(pData,SizeOfEntry,pMemory,SizeOfMemory);
END_METHOD

METHOD PUBLIC dequeueStream : BOOL //TRUE if method was successful
VAR_INPUT
	pData													: 	POINTER TO BYTE := 0;
	SizeOfStream											: 	UDINT := 0;
	pMemory													: 	POINTER TO BYTE := 0;
	SizeOfMemory											: 	UDINT := 0;
END_VAR
DequeueStream := SUPER^._DequeueStream(pData,SizeOfStream,pMemory,SizeOfMemory);
END_METHOD

METHOD PUBLIC enqueue : BOOL //TRUE if method was successful
VAR_INPUT
	pData													: 	POINTER TO BYTE := 0;
	SizeOfData												: 	UDINT := 0;
	pMemory													: 	POINTER TO BYTE := 0;
	SizeOfMemory											: 	UDINT := 0;
END_VAR
Enqueue := SUPER^._Enqueue(pData,SizeOfData,pMemory,SizeOfMemory);
END_METHOD

METHOD PUBLIC enqueueStream : BOOL //TRUE if method was successful
VAR_INPUT
	pData													: 	POINTER TO BYTE := 0;
	SizeOfData												: 	UDINT := 0;
	SizeOfStream											: 	UDINT := 0;
	pMemory													: 	POINTER TO BYTE := 0;
	SizeOfMemory											: 	UDINT := 0;
END_VAR
EnqueueStream := SUPER^._EnqueueStream(pData,SizeOfData,SizeOfStream,pMemory,SizeOfMemory);
END_METHOD

//Check wheter a value already exist
METHOD PUBLIC isEnqueued : uDINT //data exist in Fifo if reurn value <> 0, returns index of entry in buffer 
VAR_INPUT
	pData													: 	POINTER TO BYTE := 0;
	SizeOfData												: 	UDINT := 0;
	pMemory													: 	POINTER TO BYTE := 0;
	SizeOfMemory											: 	UDINT := 0;
END_VAR	
VAR
	i 														: 	DINT;
END_VAR
IsEnqueued := SUPER^._IsEnqueued(pData,SizeOfEntry,pMemory,SizeOfMemory);
END_METHOD

//Check wheter a value will be the next output of the buffer
METHOD PUBLIC isNextEntry : BOOL //Inputs value is the next output 
VAR_INPUT
	pData													: 	POINTER TO BYTE := 0;
	SizeOfData												: 	UDINT := 0;
	pMemory													: 	POINTER TO BYTE := 0;
	SizeOfMemory											: 	UDINT := 0;
END_VAR
VAR
END_VAR
IsNextEntry := SUPER^._IsNextEntry(pData,SizeOfEntry,pMemory,SizeOfMemory);
END_METHOD

METHOD PUBLIC readEntry : BOOL //TRUE if method was successful
VAR_INPUT
	idx														:	UDINT;
	pData													: 	POINTER TO BYTE := 0;
	SizeOfData												: 	UDINT := 0;
	pMemory													: 	POINTER TO BYTE := 0;
	SizeOfMemory											: 	UDINT := 0;
END_VAR
ReadEntry := SUPER^._ReadEntry(idx,pData,SizeOfEntry,pMemory,SizeOfMemory);
END_METHOD

//Reset complete Fifo
METHOD PUBLIC reset : BOOL //TRUE if method is finnished
VAR_INPUT
	pMemory													: 	POINTER TO BYTE := 0;
	SizeOfMemory											: 	UDINT := 0;
END_VAR
reset := SUPER^._reset(pMemory,SizeOfMemory);
END_METHOD

END_FUNCTION_BLOCK

// POUs/DataBuffer/LiFo/LiFoBase
//LiFo basic control template with external memory - based on Ringbuffer  
FUNCTION_BLOCK LiFoBase
VAR_INPUT	
	Overwrite												:	BOOL := FALSE; // TRUE = overwrite oldest entry 
END_VAR
VAR_OUTPUT
	Count													:	UDINT := 0; 	// Number of entrys	
	Full													:	BOOL ;		// TRUE when max number of entrys reached
	Empty													:	BOOL := TRUE; // TRUE when no entrys present
	ReadIdx													: 	UDINT := 0;	// Index to read newest data, will be updated to write idx with a new entry
	WriteIdx												: 	UDINT := 0;	// Last written index
END_VAR    
VAR
	Interlock												:	BOOL; 
	MaxEntrys												:	UDINT; //Maximum number of entrys based on size of data and size of memory
	SizeOfEntry												:	UDINT;
	NoOfStreamEntrys										:	UDINT;
END_VAR

;

METHOD PROTECTED _dequeue : BOOL //TRUE if method was successful
VAR_INPUT
	pData													: 	POINTER TO BYTE := 0; //pointer to destination of data
	SizeOfData												: 	UDINT := 0; //Size of destination data
	pMemory													: 	POINTER TO BYTE := 0;
	SizeOfMemory											: 	UDINT := 0;
END_VAR
IF 	pData = 0
	OR SizeOfData = 0
	OR pMemory = 0
	OR SizeOfMemory = 0
	OR Empty
THEN
	_dequeue												:= FALSE;
	RETURN;
ELSIF TestAndSet(Interlock)
THEN	
	IF Count > 0
	THEN 		
		MEMCPY(pData,pMemory + MAX(0, ReadIdx - 1) * SizeOfData,SizeOfData);
		ReadIdx												:= ReadIdx - 1;
		IF ReadIdx = 0
		THEN
			ReadIdx											:= MaxEntrys;
		END_IF
		WriteIdx											:= ReadIdx; //Reset WriteIdx to ReadIdx to start writing from there
		Count 												:= MAX(0,Count - 1);
		Empty 												:= Count = 0;
		Full												:= FALSE;
		
		_dequeue											:= TRUE;	
	ELSE 
		_dequeue											:= FALSE;
	END_IF
	
	Interlock												:= FALSE;
ELSE
	_dequeue												:= FALSE;
END_IF
END_METHOD

METHOD PROTECTED _dequeueStream : BOOL //TRUE if method was successful
VAR_INPUT
	pData													: 	POINTER TO BYTE := 0; //pointer to destination of data
	SizeOfStream											: 	UDINT := 0; //Size of destination data
	pMemory													: 	POINTER TO BYTE := 0;
	SizeOfMemory											: 	UDINT := 0;
END_VAR
VAR
	i														:	INT;
END_VAR
IF 	pData = 0
	OR SizeOfEntry = 0
	OR pMemory = 0
	OR SizeOfMemory = 0
	OR Empty 
	OR SizeOfStream > SizeOfMemory
THEN
	_dequeueStream											:= FALSE;
	RETURN;
ELSIF TestAndSet(Interlock)
THEN	
	NoOfStreamEntrys										:= (SizeOfStream / SizeOfEntry); 
	IF Count > 0  
	THEN 
		FOR i := 1 TO TO_INT(NoOfStreamEntrys)
		DO
			Interlock										:= FALSE; //To allow execution of _dequeue
			_dequeue(
				pData			:= pData + (TO_UDINT(i - 1) * SizeOfEntry),
				SizeOfData		:= SizeOfEntry,						
				pMemory			:= pMemory,									
				SizeOfMemory	:= SizeOfMemory);	
			IF Count <= 0
			THEN 
				EXIT;
			END_IF	
		END_FOR				
		_dequeueStream										:= TRUE;			
	ELSE 
		_dequeueStream										:= FALSE;
	END_IF
	
	Interlock												:= FALSE;
ELSE
	_dequeueStream											:= FALSE;
END_IF
END_METHOD

METHOD PROTECTED _enqueue : BOOL //TRUE if method was successful
VAR_INPUT
	pData													: 	POINTER TO BYTE := 0;
	SizeOfData												: 	UDINT := 0;
	pMemory													: 	POINTER TO BYTE := 0;
	SizeOfMemory											: 	UDINT := 0;
END_VAR
IF pData = 0
	OR SizeOfData = 0
	OR pMemory = 0
	OR SizeOfMemory = 0
	OR Full AND NOT Overwrite
THEN
	_Enqueue												:= FALSE;
	RETURN;
ELSIF TestAndSet(Interlock)
THEN			
	_Enqueue												:= FALSE;
	
	(* maximum count *)
	MaxEntrys 												:= (SizeOfMemory / SizeOfData);

	IF Count < MaxEntrys OR Overwrite
	THEN
		SizeOfEntry											:= SizeOfData;
		WriteIdx											:= WriteIdx + 1;	
		IF WriteIdx > TO_UDINT(MaxEntrys)
		THEN
			WriteIdx										:= 1;
		END_IF
		Readidx												:= WriteIdx; //Update Readidx to last write idx
	
		MEMCPY(pMemory + ((MAX(0,WriteIdx) - 1) * SizeOfData) ,pData,SizeOfData);		
		Count												:= MIN(Count + 1,  MaxEntrys);
		Full												:= Count >= MaxEntrys;
		Empty 												:= FALSE;	
		_Enqueue											:= TRUE;
	END_IF
	
	Interlock												:= FALSE;
ELSE
	_Enqueue												:= FALSE;
END_IF
END_METHOD

METHOD PROTECTED _enqueueStream : BOOL //TRUE if method was successful
VAR_INPUT
	pData													: 	POINTER TO BYTE := 0;
	SizeOfData												: 	UDINT ; //Size of one entry
	SizeOfStream											: 	UDINT := 0;
	pMemory													: 	POINTER TO BYTE := 0;
	SizeOfMemory											: 	UDINT := 0;
END_VAR
VAR
	cbData													: 	UDINT := 0;	
END_VAR
IF pData = 0
	OR SizeOfData = 0
	OR pMemory = 0
	OR SizeOfMemory = 0
	OR SizeOfStream = 0
	OR SizeOfStream > SizeOfMemory 
THEN
	_EnqueueStream											:= FALSE;
	RETURN;
ELSIF TestAndSet(Interlock)
THEN			
	_EnqueueStream											:= FALSE;
	
	(* maximum count *)
	MaxEntrys 												:= (SizeOfMemory / SizeOfData);
	SizeOfEntry												:= SizeOfData;
	NoOfStreamEntrys										:= (SizeOfStream / SizeOfData);
	
	IF (WriteIdx) + NoOfStreamEntrys <= MaxEntrys
	THEN //write full stream
		IF Count < MaxEntrys OR Overwrite
		THEN
			IF MaxEntrys = Count
			THEN //Adapt read index if write index is in front of read index
				ReadIdx										:= ReadIdx + TO_UDINT(NoOfStreamEntrys); 			
			END_IF		
		
			MEMCPY(pMemory + (WriteIdx * SizeOfData) ,pData,SizeOfStream);		
			WriteIdx										:= writeIdx + TO_UDINT(NoOfStreamEntrys);
	
			Count											:= MIN(Count + NoOfStreamEntrys, MaxEntrys);
			Empty 											:= FALSE;	
			_EnqueueStream									:= TRUE;
		ELSE
			_EnqueueStream									:= FALSE;
		END_IF	
	ELSIF Count + NoOfStreamEntrys <= (MaxEntrys) OR Overwrite
	THEN //Stream causes overflow
		cbData												:= TO_UDINT(MaxEntrys) - WriteIdx; 		 
		//Copy first part of stream to fill up buffer
		MEMCPY(pMemory + (WriteIdx * SizeOfData) ,pData, (cbData * SizeOfData) );	
		//Copy second part of stream to beginning of buffer
		MEMCPY(pMemory , pData + (cbData * SizeOfData) ,(TO_UDINT(NoOfStreamEntrys) - cbData) * SizeOfData);	
		
		WriteIdx											:= (writeIdx + TO_UDINT(NoOfStreamEntrys)) - TO_UDINT(MaxEntrys);
		Count												:= MIN(Count + NoOfStreamEntrys, MaxEntrys);
		IF MaxEntrys = Count
		THEN //Adapt read index if write index is in front of read index
			ReadIdx											:= WriteIdx;
		END_IF	
		
		Empty 												:= FALSE;	
		_EnqueueStream										:= TRUE;	
	ELSE
		_EnqueueStream										:= FALSE;	
	END_IF		
	Full													:= Count >= MaxEntrys;
	Interlock												:= FALSE;
ELSE
	_EnqueueStream											:= FALSE;
END_IF
END_METHOD

//Check wheter a value already exist
METHOD PROTECTED _isEnqueued : UDINT //data exist in Fifo if reurn value <> 0, returns index of entry in buffer 
VAR_INPUT
	pData													: 	POINTER TO BYTE := 0;
	SizeOfData												: 	UDINT := 0;
	pMemory													: 	POINTER TO BYTE := 0;
	SizeOfMemory											: 	UDINT := 0;
END_VAR	
VAR
	i,j 													: 	UDINT;
END_VAR
IF 	pData = 0
	OR SizeOfData = 0
	OR pMemory = 0
	OR SizeOfMemory = 0
	OR Empty
THEN
	_IsEnqueued												:= 0;
	RETURN;
ELSIF TestAndSet(Interlock)
THEN	
	_IsEnqueued												:= 0;
	MaxEntrys 												:= SizeOfMemory / SizeOfData;
	j														:= Writeidx;
	FOR i := Count TO 1
	DO
		IF MEMCMP(pData,pMemory + ((j - 1) * SizeOfData), SizeOfData) = 0
		THEN
			_isEnqueued										:= j;
			EXIT;
		END_IF
		j													:= j - 1;
		IF j <= 0
		THEN
			j												:= MaxEntrys;
		END_IF
	END_FOR
	Interlock												:= FALSE;
END_IF
END_METHOD

//Check wheter a value will be the next output of the buffer
METHOD PROTECTED _isNextEntry : BOOL //Inputs value is the next output 
VAR_INPUT
	pData													: 	POINTER TO BYTE := 0;
	SizeOfData												: 	UDINT := 0;
	pMemory													: 	POINTER TO BYTE := 0;
	SizeOfMemory											: 	UDINT := 0;
END_VAR
VAR
END_VAR
_IsNextEntry 	:= 0 = MEMCMP(pData,pMemory +(TO_UDINT(WriteIdx -1) * SizeOfData), SizeOfData) and NOT Empty;
END_METHOD

METHOD PROTECTED _readEntry : BOOL //TRUE if method was successful
VAR_INPUT
	idx														:	UDINT;
	pData													: 	POINTER TO BYTE := 0;
	SizeOfData												: 	UDINT := 0;
	pMemory													: 	POINTER TO BYTE := 0;
	SizeOfMemory											: 	UDINT := 0;
END_VAR
IF 	pData = 0
	OR SizeOfData = 0
	OR pMemory = 0
	OR SizeOfMemory = 0
	OR Empty
THEN
	_ReadEntry												:= FALSE;
	RETURN;
ELSIF TestAndSet(Interlock)
THEN	
	MaxEntrys 												:= SizeOfMemory / SizeOfData;
	IF idx < 1 OR idx > MIN(Count,MaxEntrys)
	THEN
		_ReadEntry											:= FALSE;
	ELSE
		MEMCPY(pData,pMemory + ((idx - 1) * SizeOfData), SizeOfData);
		_ReadEntry											:= TRUE;					
	END_IF
	Interlock												:= FALSE;
END_IF
END_METHOD

//Reset complete Fifo
METHOD PROTECTED _reset : BOOL //TRUE if method is finnished
VAR_INPUT
	pMemory													: 	POINTER TO BYTE := 0;
	SizeOfMemory											: 	UDINT := 0;
END_VAR
IF pMemory = 0
	OR SizeOfMemory = 0
THEN
	_reset													:= FALSE;
	RETURN;
ELSIF TestAndSet(Interlock)
THEN
	(* delete *)
	_reset													:= TRUE;
	MEMSET(pMemory,0,SizeOfMemory);
	ReadIdx := WriteIdx										:= 0;
	Empty 													:= TRUE;
	Full													:= FALSE;
	Count 													:= 0;
	Interlock												:= FALSE;
ELSE
	_reset													:= TRUE;
END_IF
END_METHOD

END_FUNCTION_BLOCK

// POUs/DataBuffer/Ringbuffer/Ringbuffer
//Ringbuffer based on external memory
FUNCTION_BLOCK Ringbuffer EXTENDS RingbufferBase
VAR_INPUT	
END_VAR
VAR_OUTPUT
END_VAR    
VAR
END_VAR

METHOD PUBLIC dequeue : BOOL //TRUE if method was successful
VAR_INPUT
	pData													: 	POINTER TO BYTE ;
	SizeOfData												: 	UDINT ;
	pMemory													: 	POINTER TO BYTE ;
	SizeOfMemory											: 	UDINT ;
END_VAR
Dequeue := SUPER^._Dequeue(pData,SizeOfData,pMemory,SizeOfMemory);
END_METHOD

METHOD PUBLIC dequeueStream : BOOL //TRUE if method was successful
VAR_INPUT
	pData													: 	POINTER TO BYTE ;
	SizeOfStream											:	UDINT ; //n * Size of last entry and not greater than SizeOfMemory
	pMemory													: 	POINTER TO BYTE;
	SizeOfMemory											: 	UDINT ;
END_VAR
VAR
END_VAR
DequeueStream := SUPER^._DequeueStream(pData,SizeOfStream,pMemory,SizeOfMemory);
END_METHOD

METHOD PUBLIC enqueue : BOOL //TRUE if method was successful
VAR_INPUT
	pData													: 	POINTER TO BYTE ;
	SizeOfData												: 	UDINT ;
	pMemory													: 	POINTER TO BYTE ;
	SizeOfMemory											: 	UDINT ;
END_VAR
Enqueue := SUPER^._Enqueue(pData,SizeOfData,pMemory,SizeOfMemory);
END_METHOD

METHOD PUBLIC enqueueStream : BOOL
VAR_INPUT
	pData													: 	POINTER TO BYTE ;
	SizeOfData												: 	UDINT ; //Size of one entry
	SizeOfStream											:	UDINT ; //n * SizeofData and not greater than SizeOfMemory
	pMemory													: 	POINTER TO BYTE ;
	SizeOfMemory											: 	UDINT ;
END_VAR
VAR
END_VAR
EnqueueStream := SUPER^._EnqueueStream(pData,SizeOfData,SizeOfStream,pMemory,SizeOfMemory);
END_METHOD

//Reset complete ring buffer
METHOD PUBLIC reset : BOOL //TRUE if method is finnished
VAR_INPUT
	pMemory													: 	POINTER TO BYTE := 0;
	SizeOfMemory											: 	UDINT := 0;
END_VAR
reset := SUPER^._reset(pMemory,SizeOfMemory);
END_METHOD

END_FUNCTION_BLOCK

// POUs/DataBuffer/Ringbuffer/RingbufferBase
//Ringbuffer basic template based on external memory
FUNCTION_BLOCK RingbufferBase
VAR_INPUT	
	Overwrite												:	BOOL := FALSE; // TRUE = overwrite oldest entry 
END_VAR
VAR_OUTPUT
	Count													:	UDINT := 0; 	// Number of entrys	
	Full													:	BOOL ;		// TRUE when max number of entrys reached
	Empty													:	BOOL := TRUE; // TRUE when no entrys present
	ReadIdx													: 	UDINT := 0;	// Read idx, starting from oldest entry
	WriteIdx												: 	UDINT := 0;	// Write idx 
END_VAR    
VAR
	Interlock												:	BOOL; 
	MaxEntrys												:	UDINT; //Maximum number of entrys based on size of data and size of memory
	SizeOfEntry												:	UDINT;
	NoOfStreamEntrys										:	UDINT;
	cbData													:	UDINT;
END_VAR

METHOD PROTECTED _dequeue : BOOL //TRUE if method was successful - copies oldest entry and set ReadIdx 
VAR_INPUT
	pData													: 	POINTER TO BYTE ;
	SizeOfData												: 	UDINT ;
	pMemory													: 	POINTER TO BYTE ;
	SizeOfMemory											: 	UDINT ;
END_VAR
IF 	pData = 0
	OR SizeOfData = 0
	OR pMemory = 0
	OR SizeOfMemory = 0
	OR Empty
THEN
	_Dequeue												:= FALSE;
	RETURN;
ELSIF TestAndSet(Interlock)
THEN	
	IF Count > 0
	THEN 
		(* copy dataset *)
		ReadIdx												:= ReadIdx + 1;
		IF (ReadIdx) > MaxEntrys
		THEN
			ReadIdx											:= 1;						
		END_IF
		
		MEMCPY(pData,pMemory + MAX(0, ReadIdx - 1) * SizeOfData,SizeOfData);
		
		Count 												:= MAX(0,Count - 1);
		Empty 												:= Count = 0;
		Full												:= FALSE;
		_Dequeue											:= TRUE;	
	ELSE 
		_Dequeue											:= FALSE;
	END_IF
	
	Interlock												:= FALSE;
ELSE
	_Dequeue												:= FALSE;
END_IF
END_METHOD

METHOD PROTECTED _dequeueStream : BOOL //TRUE if method was successful - copies oldest data and set ready index 
VAR_INPUT
	pData													: 	POINTER TO BYTE ;
	SizeOfStream											:	UDINT ; //n * Size of last entry and not greater than SizeOfMemory
	pMemory													: 	POINTER TO BYTE;
	SizeOfMemory											: 	UDINT ;
END_VAR
VAR
END_VAR
IF 	pData = 0
	OR SizeOfEntry = 0
	OR pMemory = 0
	OR SizeOfMemory = 0
	OR Empty 
	OR SizeOfStream > SizeOfMemory
THEN
	_DequeueStream											:= FALSE;
	RETURN;
ELSIF TestAndSet(Interlock)
THEN	
	NoOfStreamEntrys										:= (SizeOfStream / SizeOfEntry); 
	IF Count > 0  
	THEN 
		(* maximum count *)
		IF ReadIdx + MIN(Count,NoOfStreamEntrys) <= MaxEntrys
		THEN //Read all data at one time
			ReadIdx											:= ReadIdx + 1; //Point to start read data			
			MEMCPY(pData,pMemory + (ReadIdx - 1) * SizeOfEntry, MIN(TO_UDINT(Count) * SizeOfEntry, SizeOfStream));
			ReadIdx											:= (ReadIdx - 1) + TO_UDINT(MIN(Count, NoOfStreamEntrys)); //Point to next index after reading x entrys
				
		ELSE //Read data with overflow					
			cbData											:= TO_UDINT(MaxEntrys) - ReadIdx; 		 
			ReadIdx											:= ReadIdx + 1; //Point to start read data	
			//Copy first part of stream our from buffer
			MEMCPY(pData, pMemory + ((ReadIdx - 1) * SizeOfEntry), cbData * SizeOfEntry );
	
			//Copy second part of stream from beginning of buffer
			ReadIdx											:= TO_UDINT(MIN(Count,NoOfStreamEntrys)) - cbData; //Point to next index after reading x entrys	
			MEMCPY( pData + (cbData * SizeOfEntry) , pMemory ,(TO_UDINT(MIN(Count,NoOfStreamEntrys)) - cbData) * SizeOfEntry);			
		END_IF
		Count 												:= MAX(0,Count - NoOfStreamEntrys);		
		Empty 												:= Count = 0;
		Full												:= FALSE;
		_DequeueStream										:= TRUE;	
		
	ELSE 
		_DequeueStream										:= FALSE;
	END_IF
	
	Interlock												:= FALSE;
ELSE
	_DequeueStream											:= FALSE;
END_IF
END_METHOD

METHOD PROTECTED _enqueue : BOOL //TRUE if method was successful
VAR_INPUT
	pData													: 	POINTER TO BYTE ;
	SizeOfData												: 	UDINT ;
	pMemory													: 	POINTER TO BYTE ;
	SizeOfMemory											: 	UDINT ;
END_VAR
IF pData = 0
	OR SizeOfData = 0
	OR pMemory = 0
	OR SizeOfMemory = 0
THEN
	_Enqueue												:= FALSE;
	RETURN;
ELSIF TestAndSet(Interlock)
THEN			
	_Enqueue												:= FALSE;
	
	(* maximum count *)
	MaxEntrys 												:= (SizeOfMemory / SizeOfData);

	IF Count < MaxEntrys OR Overwrite
	THEN
		SizeOfEntry											:= SizeOfData;
		IF MaxEntrys = Count 
		THEN //Adapt read index if write index is in front of read index
			ReadIdx											:= ReadIdx + 1;
			IF ReadIdx > TO_UDINT(MaxEntrys)
			THEN
				ReadIdx										:= 1;								
			END_IF
		END_IF	
		WriteIdx											:= WriteIdx + 1;	
		IF WriteIdx > TO_UDINT(MaxEntrys)
		THEN
			WriteIdx										:= 1;
		END_IF
	
		MEMCPY(pMemory + ((MAX(0,WriteIdx) - 1) * SizeOfData) ,pData,SizeOfData);		
	
		Count												:= MIN(Count + 1,  MaxEntrys);
		Full												:= Count >= MaxEntrys;
		Empty 												:= FALSE;	
		_Enqueue											:= TRUE;
	END_IF
	
	Interlock												:= FALSE;
ELSE
	_Enqueue												:= FALSE;
END_IF
END_METHOD

METHOD PROTECTED _enqueueStream : BOOL
VAR_INPUT
	pData													: 	POINTER TO BYTE ;
	SizeOfData												: 	UDINT ; //Size of one entry
	SizeOfStream											:	UDINT ; //n * SizeofData and not greater than SizeOfMemory
	pMemory													: 	POINTER TO BYTE ;
	SizeOfMemory											: 	UDINT ;
END_VAR
VAR
END_VAR
IF pData = 0
	OR SizeOfData = 0
	OR pMemory = 0
	OR SizeOfMemory = 0
	OR SizeOfStream = 0
	OR SizeOfStream > SizeOfMemory 
THEN
	_EnqueueStream											:= FALSE;
	RETURN;
ELSIF TestAndSet(Interlock)
THEN			
	_EnqueueStream											:= FALSE;
	
	(* maximum count *)
	MaxEntrys 												:= (SizeOfMemory / SizeOfData);
	SizeOfEntry												:= SizeOfData;
	NoOfStreamEntrys										:= (SizeOfStream / SizeOfData);
	
	IF (WriteIdx) + NoOfStreamEntrys <= MaxEntrys
	THEN //write full stream
		IF Count < MaxEntrys OR Overwrite
		THEN
			IF MaxEntrys = Count
			THEN //Adapt read index if write index is in front of read index
				ReadIdx										:= ReadIdx + TO_UDINT(NoOfStreamEntrys); 			
			END_IF		
		
			MEMCPY(pMemory + (WriteIdx * SizeOfData) ,pData,SizeOfStream);		
			WriteIdx										:= writeIdx + TO_UDINT(NoOfStreamEntrys);
			
			Count											:= MIN(Count + NoOfStreamEntrys, MaxEntrys);
			Empty 											:= FALSE;	
			_EnqueueStream									:= TRUE;
		ELSE
			_EnqueueStream									:= FALSE;
		END_IF	
	ELSIF Count + NoOfStreamEntrys <= (MaxEntrys) OR Overwrite
	THEN //Stream causes overflow
		cbData												:= TO_UDINT(MaxEntrys) - WriteIdx; 		 
		//Copy first part of stream to fill up buffer
		MEMCPY(pMemory + (WriteIdx * SizeOfData) ,pData, (cbData * SizeOfData) );	
		//Copy second part of stream to beginning of buffer
		MEMCPY(pMemory , pData + (cbData * SizeOfData) ,(TO_UDINT(NoOfStreamEntrys) - cbData) * SizeOfData);	
		
		WriteIdx											:= (writeIdx + TO_UDINT(NoOfStreamEntrys)) - TO_UDINT(MaxEntrys);
		Count												:= MIN(Count + NoOfStreamEntrys, MaxEntrys);
		IF MaxEntrys = Count
		THEN //Adapt read index if write index is in front of read index
			ReadIdx											:= WriteIdx;
		END_IF	
		
		Empty 												:= FALSE;	
		_EnqueueStream										:= TRUE;	
	ELSE
		_EnqueueStream										:= FALSE;	
	END_IF		
	Full													:= Count >= MaxEntrys;
	Interlock												:= FALSE;
ELSE
	_EnqueueStream											:= FALSE;
END_IF
END_METHOD

//Reset complete ring buffer
METHOD PROTECTED _reset : BOOL //TRUE if method is finnished
VAR_INPUT
	pMemory													: 	POINTER TO BYTE := 0;
	SizeOfMemory											: 	UDINT := 0;
END_VAR
IF pMemory = 0
	OR SizeOfMemory = 0
THEN
	_reset													:= TRUE;
	RETURN;
ELSIF TestAndSet(Interlock)
THEN
	(* delete *)
	_reset													:= TRUE;
	MEMSET(pMemory,0,SizeOfMemory);
	ReadIdx := WriteIdx										:= 0;
	Empty 													:= TRUE;
	Full													:= FALSE;
	Count 													:= 0;
	Interlock												:= FALSE;
ELSE
	_reset													:= TRUE;
END_IF
END_METHOD

END_FUNCTION_BLOCK

// POUs/DataBuffer/LiFo/LiFoExt
//LifoBase extended with dynamical memory allocation
 {attribute 'enable_dynamic_creation'}
FUNCTION_BLOCK LiFoExt EXTENDS LiFoBase
VAR_OUTPUT CONSTANT
END_VAR   
VAR_INPUT
	MaxNoOfEntrys											: 	UDINT := 10;	//0 = dynamically allocation / <> 0 = pre allcoation of memory based on size of first entry (n * data size) 
END_VAR
VAR_OUTPUT
	pMemory													: 	POINTER TO BYTE := 0; //Pointer to memory	
	SizeOfMemory											: 	UDINT := 0; //According MaxNoOfEntrys and SizeOfData of first entry
END_VAR
VAR
	MemSizeAllocatedMemory									:	UDINT := 0; //Allocated memory 
	MemSizeOfData											:	UDINT;
	MemMaxNoOfEntrys										:	UDINT;
	ExtInterlock											:	BOOL;
END_VAR

;

METHOD PROTECTED FINAL allocate : BOOL
VAR_IN_OUT
	SizeOfData												:	UDINT;
END_VAR
VAR
	pDummy													:	POINTER TO BYTE;	
End_Var
IF pMemory = 0
THEN
	IF SizeOfData = 0 OR MaxNoOfEntrys = 0
	THEN
		Allocate											:= FALSE;	
	ELSE
		MemSizeOfData										:= SizeOfData;
		MemMaxNoOfEntrys									:= MaxNoOfEntrys;
		SizeOfMemory										:= MemSizeOfData * MemMaxNoOfEntrys;
		MemSizeAllocatedMemory								:= SizeOfMemory;
		pMemory												:= __NEW(BYTE,SizeOfMemory );
		
		IF PARAM.ENABLE_DEBUG_MSG_DYNAMIC_MEM_ALLOCATION
		THEN
			AdsLogHint('EngineeringToolbox | FB FifoExt | An instance allocated %s bytes from the dynamic memory of the ADS router memory pool', TO_STRING(SizeOfMemory));
		END_IF
	END_IF

ELSIF SizeOfData = MemSizeOfData AND MaxNoOfEntrys = MemMaxNoOfEntrys
THEN
	Allocate												:= TRUE;
	
ELSIF SizeOfData > MemSizeOfData OR MaxNoOfEntrys > MemMaxNoOfEntrys
THEN //Since increased, allocate new memory
	MemSizeAllocatedMemory									:= SizeOfData * MaxNoOfEntrys;
	pDummy													:= __NEW(BYTE, MemSizeAllocatedMemory); 
	
	 //Size of data still the same, copy old data to reuse
	IF MemSizeOfData = SizeOfData AND Count > 0
	THEN
		MEMCPY(pDummy,pMemory, SizeOfMemory);
	END_IF
	
	//Copy new settings to local variales
	MemSizeOfData											:= SizeOfData;
	MemMaxNoOfEntrys										:= MaxNoOfEntrys;	
	SizeOfMemory 											:= MemSizeAllocatedMemory;

	__DELETE(pMemory);  //Delete reference to old memory
	pMemory													:= pDummy; //Take over new pointer to new memory
	
	IF PARAM.ENABLE_DEBUG_MSG_DYNAMIC_MEM_ALLOCATION
	THEN
		AdsLogWarn('EngineeringToolbox | FB FifoExt | Value of "MaxNoOfEntrys" or data size increased and one instance allocated additional %s bytes from the dynamic memory of the ADS router memory pool', TO_STRING(SizeOfMemory));
	END_IF
	
	Allocate												:= TRUE;
	
ELSE //Size decreased
	IF MemSizeOfData <> SizeOfData AND Count > 0
	THEN //Size of data changed, erease memory 
		MEMSET(pMemory,0, MemSizeAllocatedMemory);
	ELSE //Size of data the same, keep current data
		;
	END_IF
	
	//Copy new settings to local variales
	MemSizeOfData											:= SizeOfData;
	MemMaxNoOfEntrys										:= MaxNoOfEntrys;
	SizeOfMemory											:= MemSizeOfData * MemMaxNoOfEntrys;
	Allocate												:= TRUE;
END_IF
END_METHOD

METHOD PUBLIC dequeue : BOOL //TRUE if method was successful
VAR_INPUT
	pData													:	POINTER TO BYTE;	
END_VAR
VAR
END_VAR
Dequeue := SUPER^._Dequeue(pData,SizeOfEntry,This^.pMemory,This^.SizeOfMemory);
END_METHOD

METHOD PUBLIC dequeueStream : BOOL //TRUE if method was successful
VAR_INPUT
	pData													: 	POINTER TO BYTE := 0;
	SizeOfStream											: 	UDINT := 0;
	pMemory													: 	POINTER TO BYTE := 0;
	SizeOfMemory											: 	UDINT := 0;
END_VAR
DequeueStream := SUPER^._DequeueStream(pData,SizeOfStream,pMemory,SizeOfMemory);
END_METHOD

METHOD PUBLIC enqueue : BOOL //TRUE if method was successful
VAR_INPUT
	pData													:	POINTER TO BYTE;
	SizeOfData												:	UDINT;
END_VAR
VAR
	CopySize												:	UDINT;
	pDummy													:	POINTER TO BYTE;
END_VAR
IF TestAndSet(ExtInterlock) 
THEN	
	if Allocate(SizeOfData)
	then
		Enqueue 											:= SUPER^._Enqueue(pData,SizeOfData,THIS^.pMemory,THIS^.SizeOfMemory);
		ExtInterlock										:= FALSE;
	else
		Enqueue												:= FALSE;
	END_IF	
ELSE
	Enqueue													:= FALSE;
END_IF
END_METHOD

METHOD PUBLIC enqueueStream : BOOL //TRUE if method was successful
VAR_INPUT
	pData													: 	POINTER TO BYTE := 0;
	SizeOfData												: 	UDINT := 0;
	SizeOfStream											: 	UDINT := 0;
	pMemory													: 	POINTER TO BYTE := 0;
	SizeOfMemory											: 	UDINT := 0;
END_VAR
EnqueueStream := SUPER^._EnqueueStream(pData,SizeOfData, SizeOfStream,pMemory,SizeOfMemory);
END_METHOD

METHOD FB_exit : BOOL
VAR_INPUT
	bInCopyCode : BOOL; // if TRUE, the exit method is called for exiting an instance that is copied afterwards (online change).
END_VAR
IF NOT bInCopyCode AND pMemory <> 0
THEN //Release memory in case the PLC stopps
	__DELETE(pMemory);
	Full													:= FALSE;
	Empty													:= TRUE;
	Count													:= 0;
	SizeOfMemory											:= 0;
	MemSizeOfData											:= 0;
	MemSizeAllocatedMemory									:= 0;
	MemMaxNoOfEntrys										:= MaxNoOfEntrys;
END_IF
END_METHOD

//Check wheter a value already exist
METHOD PUBLIC isEnqueued : UDINT //pData entry exist in Fifo at idx as return value 
VAR_INPUT
	pData													: 	POINTER TO BYTE := 0;
END_VAR
IsEnqueued := SUPER^._IsEnqueued(pData,SizeOfEntry,This^.pMemory,This^.SizeOfMemory);
END_METHOD

//Check wheter a value will be the next output of the buffer
METHOD PUBLIC isNextEntry : BOOL //Inputs value is the next output 
VAR_INPUT
	pData													: 	POINTER TO BYTE := 0;
END_VAR
VAR
END_VAR
IsNextEntry := SUPER^._IsNextEntry(pData,SizeOfEntry,This^.pMemory,This^.SizeOfMemory);
END_METHOD

METHOD PUBLIC readEntry : BOOL //TRUE if method was successful
VAR_INPUT
	idx														:	UDINT;
	pData													: 	POINTER TO BYTE := 0;
END_VAR
ReadEntry := SUPER^._ReadEntry(idx,pData,SizeOfEntry,This^.pMemory,This^.SizeOfMemory);
END_METHOD

//Reset complete Fifo
METHOD PUBLIC reset : BOOL //TRUE if method is finnished
VAR_INPUT
END_VAR
reset				:= SUPER^._reset(This^.pMemory,This^.SizeOfMemory);
END_METHOD

END_FUNCTION_BLOCK

// POUs/DataBuffer/Ringbuffer/RingbufferByteSimple
//Ringbuffer with a internal Byte array for a simple data buffer implementation 
FUNCTION_BLOCK RingbufferByteSimple EXTENDS RingbufferBase
VAR_OUTPUT CONSTANT
	MIN_BUFFER												:	UDINT := 1; //Ringbuffer start index 
	MAX_BUFFER												:	uDINT := PARAM.RINGBUFFER_BYTE_SIMPLE_MAX_BUFFER; //Ringbuffer buffer end index - see library parameter to customize parameter
END_VAR   
VAR_INPUT
END_VAR
VAR_OUTPUT
	Buffer													:	ARRAY[MIN_BUFFER..MAX_BUFFER] OF BYTE; //Byte buffer 
END_VAR
VAR 
END_VAR

;

METHOD PUBLIC dequeue : BOOL //TRUE if method was successful
VAR_IN_OUT
	value													: BYTE;	
END_VAR
IF TestAndSet(Interlock)
THEN	
	IF Count > 0
	THEN 
		(* copy dataset *)		
		ReadIdx												:= ReadIdx + 1;
		IF (ReadIdx) > MAX_BUFFER
		THEN
			ReadIdx											:= TO_UDINT(MIN_BUFFER);				
		END_IF
		
		Value												:= Buffer[ReadIdx];
		
		Count 												:= MAX(0,Count - 1);
		Empty 												:= Count = 0;
		Full												:= FALSE;
		Dequeue												:= TRUE;	
	ELSE 
		Dequeue												:= FALSE;
	END_IF
	
	Interlock												:= FALSE;
ELSE
	Dequeue													:= FALSE;
END_IF
END_METHOD

METHOD PUBLIC dequeueStream : BOOL //TRUE if method was successful
VAR_INPUT
	pData													:	POINTER TO BYTE;
	SizeOfStream											:	UDINT;	
END_VAR
DequeueStream := super^._DequeueStream(pData, SizeOfStream,  ADR(Buffer),SIZEOF(Buffer));
END_METHOD

METHOD PUBLIC enqueue : BOOL //TRUE if method was successful
VAR_INPUT
	Value													:	BYTE;
END_VAR
IF TestAndSet(Interlock)
THEN			
	Enqueue													:= FALSE;

	IF Count < MAX_BUFFER OR Overwrite
	THEN
		IF MAX_BUFFER = Count 
		THEN //Adapt read index if write index is in front of read index
			ReadIdx											:= ReadIdx + 1;
			IF ReadIdx > TO_UDINT(MAX_BUFFER)
			THEN
				ReadIdx										:= TO_UDINT(MIN_BUFFER);							
			END_IF
		END_IF		
		WriteIdx											:= WriteIdx + 1;	
		IF WriteIdx > TO_UDINT(MAX_BUFFER)
		THEN
			WriteIdx										:= TO_UDINT(MIN_BUFFER);
		END_IF
	
		Buffer[WriteIdx]									:= Value;
	
		Count												:= MIN(Count + 1,  MAX_BUFFER);
		Full												:= Count >= MAX_BUFFER;
		Empty 												:= FALSE;	
		Enqueue												:= TRUE;
	END_IF
	
	Interlock												:= FALSE;
ELSE
	Enqueue													:= FALSE;
END_IF
END_METHOD

METHOD PUBLIC enqueueStream : BOOL //TRUE if method was successful
VAR_INPUT
	pData													:	POINTER TO BYTE;
	SizeOfStream											:	UDINT;
END_VAR
EnqueueStream := SUPER^._EnqueueStream(pData, SIZEOF(BUFFER[MIN_BUFFER] ), SizeOfStream,ADR(Buffer),SIZEOF(Buffer));
END_METHOD

//Reset complete ring buffer
METHOD PUBLIC reset : BOOL //TRUE if method is finnished
VAR_INPUT
END_VAR
reset := SUPER^._reset(ADR(Buffer),SIZEOF(Buffer));
END_METHOD

END_FUNCTION_BLOCK

// POUs/DataBuffer/Ringbuffer/RingbufferCharSimple
//Ringbuffer with a internal char array (String) for a simple num list implementation
FUNCTION_BLOCK RingbufferCharSimple EXTENDS RingbufferBase
VAR_OUTPUT CONSTANT
	MIN_BUFFER												:	UDINT := 0; //Default min index of string 
	MAX_BUFFER												:	UDINT := PARAM.RINGBUFFER_CHAR_SIMPLE_MAX_BUFFER; //Ringbuffer buffer end index - see library parameter to customize parameter
END_VAR   
VAR_INPUT
END_VAR
VAR_OUTPUT
	Buffer													:	STRING[MAX_BUFFER]; //Char buffer 
END_VAR
VAR
END_VAR

;

METHOD PUBLIC dequeue : BOOL //TRUE if method was successful
VAR_IN_OUT
	value													: BYTE;	
END_VAR
Dequeue := SUPER^._Dequeue(ADR(Value),SizeOfEntry,ADR(Buffer),SIZEOF(Buffer));
END_METHOD

METHOD PUBLIC dequeueStream : BOOL //TRUE if method was successful
VAR_INPUT
	pData													:	POINTER TO BYTE;
	SizeOfStream											:	UDINT ; //Not greater than SizeOfMemory
END_VAR
DequeueStream := SUPER^._DequeueStream(pData, SizeOfStream,  ADR(Buffer),TO_UDINT(MAX_BUFFER));
END_METHOD

METHOD PUBLIC enqueue : BOOL //TRUE if method was successful
VAR_INPUT
	Value													:	BYTE;
END_VAR
Enqueue := SUPER^._Enqueue(ADR(Value),SIZEOF(Value),ADR(Buffer),SIZEOF(Buffer));
END_METHOD

METHOD PUBLIC enqueueStream : BOOL //TRUE if method was successful
VAR_INPUT
	pData													:	POINTER TO BYTE;
	SizeOfStream											:	UDINT ; //Not greater than SizeOfMemory
END_VAR
EnqueueStream := SUPER^._EnqueueStream(pData,SIZEOF(BUFFER[MIN_BUFFER]), SizeOfStream,ADR(Buffer),TO_UDINT(MAX_BUFFER));
END_METHOD

//Reset complete ring buffer
METHOD PUBLIC reset : BOOL //TRUE if method is finnished
VAR_INPUT
END_VAR
reset := SUPER^._reset(ADR(Buffer),SIZEOF(Buffer));
END_METHOD

END_FUNCTION_BLOCK

// POUs/DataBuffer/Ringbuffer/RingbufferExt
//Ringbuffer extended with dynamical allocation of memory 
{attribute 'enable_dynamic_creation'}
FUNCTION_BLOCK RingbufferExt EXTENDS RingbufferBase
VAR_OUTPUT CONSTANT
END_VAR   
VAR_INPUT
	MaxNoOfEntrys											: 	UDINT := 10;	//0 = dynamically allocation / <> 0 = pre allcoation of memory based on size of first entry (n * data size) 
END_VAR
VAR_OUTPUT
	pMemory													: 	POINTER TO BYTE := 0;	//start address of buffer data
	SizeOfMemory											: 	UDINT := 0;	//size of buffer
END_VAR
VAR
	MemSizeAllocatedMemory									:	UDINT := 0; //Allocated memory 
	MemSizeOfData											:	UDINT;
	MemMaxNoOfEntrys										:	UDINT;
	ExtInterlock											:	BOOL;
END_VAR

;

METHOD PROTECTED FINAL allocate : BOOL
VAR_IN_OUT
	SizeOfData												:	UDINT;
END_VAR
VAR
	pDummy													:	POINTER TO BYTE;	
End_Var
IF pMemory = 0
THEN
	IF SizeOfData = 0 OR MaxNoOfEntrys = 0
	THEN
		Allocate											:= FALSE;	
	ELSE
		MemSizeOfData										:= SizeOfData;
		MemMaxNoOfEntrys									:= MaxNoOfEntrys;
		SizeOfMemory										:= MemSizeOfData * MemMaxNoOfEntrys;
		MemSizeAllocatedMemory								:= SizeOfMemory;
		pMemory												:= __NEW(BYTE,SizeOfMemory );
		
		IF PARAM.ENABLE_DEBUG_MSG_DYNAMIC_MEM_ALLOCATION
		THEN
			AdsLogHint('EngineeringToolbox | FB FifoExt | An instance allocated %s bytes from the dynamic memory of the ADS router memory pool', TO_STRING(SizeOfMemory));
		END_IF
	END_IF

ELSIF SizeOfData = MemSizeOfData AND MaxNoOfEntrys = MemMaxNoOfEntrys
THEN
	Allocate												:= TRUE;
	
ELSIF SizeOfData > MemSizeOfData OR MaxNoOfEntrys > MemMaxNoOfEntrys
THEN //Since increased, allocate new memory
	MemSizeAllocatedMemory									:= SizeOfData * MaxNoOfEntrys;
	pDummy													:= __NEW(BYTE, MemSizeAllocatedMemory); 
	
	 //Size of data still the same, copy old data to reuse
	IF MemSizeOfData = SizeOfData AND Count > 0
	THEN
		MEMCPY(pDummy,pMemory, SizeOfMemory);
	END_IF
	
	//Copy new settings to local variales
	MemSizeOfData											:= SizeOfData;
	MemMaxNoOfEntrys										:= MaxNoOfEntrys;	
	SizeOfMemory 											:= MemSizeAllocatedMemory;

	__DELETE(pMemory);  //Delete reference to old memory
	pMemory													:= pDummy; //Take over new pointer to new memory
	
	IF PARAM.ENABLE_DEBUG_MSG_DYNAMIC_MEM_ALLOCATION
	THEN
		AdsLogWarn('EngineeringToolbox | FB FifoExt | Value of "MaxNoOfEntrys" or data size increased and one instance allocated additional %s bytes from the dynamic memory of the ADS router memory pool', TO_STRING(SizeOfMemory));
	END_IF
	
	Allocate												:= TRUE;
	
ELSE //Size decreased
	IF MemSizeOfData <> SizeOfData AND Count > 0
	THEN //Size of data changed, erease memory 
		MEMSET(pMemory,0, MemSizeAllocatedMemory);
	ELSE //Size of data the same, keep current data
		;
	END_IF
	
	//Copy new settings to local variales
	MemSizeOfData											:= SizeOfData;
	MemMaxNoOfEntrys										:= MaxNoOfEntrys;
	SizeOfMemory											:= MemSizeOfData * MemMaxNoOfEntrys;
	Allocate												:= TRUE;
END_IF
END_METHOD

METHOD PUBLIC dequeue : BOOL //TRUE if method was successful
VAR_INPUT
	pData													:	POINTER TO BYTE;	
END_VAR
VAR
END_VAR
Dequeue := SUPER^._Dequeue(pData,SizeOfEntry,This^.pMemory,This^.SizeOfMemory);
END_METHOD

METHOD PUBLIC dequeueStream : BOOL //TRUE if method was successful
VAR_INPUT
	pData													:	POINTER TO BYTE;	
	SizeOfStream											:	UDINT ; //Not greater than SizeOfMemory
END_VAR
VAR
END_VAR
DequeueStream := SUPER^._DequeueStream(pData,SizeOfStream , This^.pMemory,This^.SizeOfMemory);
END_METHOD

METHOD PUBLIC enqueue : BOOL //TRUE if method was successful
VAR_INPUT
	pData													:	POINTER TO BYTE;
	SizeOfData												:	UDINT;
END_VAR
VAR
END_VAR
IF TestAndSet(ExtInterlock) 
THEN	
	if Allocate(SizeOfData)
	then
		Enqueue 											:= SUPER^._Enqueue(pData,SizeOfData,THIS^.pMemory,THIS^.SizeOfMemory);
		ExtInterlock										:= FALSE;
	else
		Enqueue												:= FALSE;
	END_IF	
ELSE
	Enqueue													:= FALSE;
END_IF
END_METHOD

METHOD PUBLIC enqueueStream : BOOL //TRUE if method was successful
VAR_INPUT
	pData													:	POINTER TO BYTE;
	SizeOfData												:	UDINT; //Size of one entry
	SizeOfStream											:	UDINT ; //Not greater than SizeOfMemory
END_VAR
VAR
END_VAR
IF TestAndSet(ExtInterlock) 
THEN	
	if Allocate(SizeOfData)
	then
		EnqueueStream 										:= SUPER^._EnqueueStream(pData,SizeOfData,SizeOfStream,THIS^.pMemory,THIS^.SizeOfMemory);
		ExtInterlock										:= FALSE;
	else
		EnqueueStream										:= FALSE;
	END_IF	
ELSE
	EnqueueStream											:= FALSE;
END_IF
END_METHOD

METHOD FB_exit : BOOL
VAR_INPUT
	bInCopyCode : BOOL; // if TRUE, the exit method is called for exiting an instance that is copied afterwards (online change).
END_VAR
IF NOT bInCopyCode AND pMemory <> 0
THEN //Release memory in case the PLC stopps
	__DELETE(pMemory);
	SizeOfMemory								:= 0;
END_IF
END_METHOD

//Reset complete ring buffer
METHOD PUBLIC reset : BOOL //TRUE if method is finnished
VAR_INPUT
END_VAR
IF pMemory = 0
THEN //no memroy allocated
	reset													:= TRUE;
ELSE //Just delte the memory
	reset 													:= SUPER^._reset(THIS^.pMemory,THIS^.SizeOfMemory);	
END_IF
END_METHOD

END_FUNCTION_BLOCK

// POUs/DataBuffer/Ringbuffer/RingbufferLRealSimple
//Ringbuffer with a internal Lreal array for a simple num list implementation 
FUNCTION_BLOCK RingbufferLRealSimple EXTENDS RingbufferBase
VAR_OUTPUT CONSTANT
	MIN_BUFFER												:	UDINT := 1; //Ringbuffer start index
	MAX_BUFFER												:	UDINT := PARAM.RINGBUFFER_LREAL_SIMPLE_MAX_BUFFER; //Ringbuffer buffer end index - see library parameter to customize parameter
END_VAR   
VAR_INPUT
END_VAR
VAR_OUTPUT
	Buffer													:	ARRAY[MIN_BUFFER..MAX_BUFFER] OF LREAL; //Lreal buffer 
END_VAR
VAR 
END_VAR

;

METHOD PUBLIC dequeue : BOOL //TRUE if method was successful
VAR_IN_OUT
	value													: LREAL;	
END_VAR
Dequeue := SUPER^._Dequeue(ADR(Value),SizeOfEntry,ADR(Buffer),SIZEOF(Buffer));
END_METHOD

METHOD PUBLIC dequeueStream : BOOL //TRUE if method was successful
VAR_INPUT
	pData													:	POINTER TO LREAL;
	SizeOfStream											:	UDINT ; //Not greater than SizeOfMemory
END_VAR
DequeueStream := super^._DequeueStream(pData,SizeOfStream,  ADR(Buffer),SIZEOF(Buffer));
END_METHOD

METHOD PUBLIC enqueue : BOOL //TRUE if method was successful
VAR_INPUT
	Value													:	LREAL;
END_VAR
Enqueue := SUPER^._Enqueue(ADR(Value),SIZEOF(Value),ADR(Buffer),SIZEOF(Buffer));
END_METHOD

METHOD PUBLIC enqueueStream : BOOL //TRUE if method was successful
VAR_INPUT
	pData													:	POINTER TO LREAL;
	SizeOfStream											:	UDINT ; //Not greater than SizeOfMemory
END_VAR
EnqueueStream := SUPER^._EnqueueStream(pData,SIZEOF(BUFFER[MIN_BUFFER]), SizeOfStream,ADR(Buffer),SIZEOF(Buffer));
END_METHOD

//Reset complete ring buffer
METHOD PUBLIC reset : BOOL //TRUE if method is finnished
VAR_INPUT
END_VAR
reset := SUPER^._reset(ADR(Buffer),SIZEOF(Buffer));
END_METHOD

END_FUNCTION_BLOCK

// POUs/DataBuffer/Ringbuffer/RingbufferRealSimple
//Ringbuffer with a internal Lreal array for a simple num list implementation 
FUNCTION_BLOCK RingbufferRealSimple EXTENDS RingbufferBase
VAR_OUTPUT CONSTANT
	MIN_BUFFER												:	UDINT := 1; //Ringbuffer start index
	MAX_BUFFER												:	UDINT := PARAM.RINGBUFFER_REAL_SIMPLE_MAX_BUFFER; //Ringbuffer buffer end index - see library parameter to customize parameter
END_VAR   
VAR_INPUT
END_VAR
VAR_OUTPUT
	Buffer													:	ARRAY[MIN_BUFFER..MAX_BUFFER] OF REAL; //Lreal buffer 
END_VAR
VAR 
END_VAR

;

METHOD PUBLIC dequeue : BOOL //TRUE if method was successful
VAR_IN_OUT
	value													: REAL;	
END_VAR
Dequeue := SUPER^._Dequeue(ADR(Value),SizeOfEntry,ADR(Buffer),SIZEOF(Buffer));
END_METHOD

METHOD PUBLIC dequeueStream : BOOL //TRUE if method was successful
VAR_INPUT
	pData													:	POINTER TO REAL;
	SizeOfStream											:	UDINT ; //Not greater than SizeOfMemory
END_VAR
DequeueStream := super^._DequeueStream(pData,SizeOfStream,  ADR(Buffer),SIZEOF(Buffer));
END_METHOD

METHOD PUBLIC enqueue : BOOL //TRUE if method was successful
VAR_INPUT
	Value													:	REAL;
END_VAR
Enqueue := SUPER^._Enqueue(ADR(Value),SIZEOF(Value),ADR(Buffer),SIZEOF(Buffer));
END_METHOD

METHOD PUBLIC enqueueStream : BOOL //TRUE if method was successful
VAR_INPUT
	pData													:	POINTER TO REAL;
	SizeOfStream											:	UDINT ; //Not greater than SizeOfMemory
END_VAR
EnqueueStream := SUPER^._EnqueueStream(pData,SIZEOF(BUFFER[MIN_BUFFER]), SizeOfStream,ADR(Buffer),SIZEOF(Buffer));
END_METHOD

//Reset complete ring buffer
METHOD PUBLIC reset : BOOL //TRUE if method is finnished
VAR_INPUT
END_VAR
reset := SUPER^._reset(ADR(Buffer),SIZEOF(Buffer));
END_METHOD

END_FUNCTION_BLOCK

// POUs/DataBuffer/DoubleBuffer
//Double buffer FB to fill one part of buffer while the other (filled) part can be read or processed meanwhile
//Variable "ReadyToRead" signals that recorded data can be read consistent by pointer "pDataToRead" 
//After the data are processed or copied, it is needed to call the method "setReadyToReady(Status := FALSE)" and release the buffer to be used if the other half is filled 
//With setReadyToReady(Status := TRUE) you can mark the current write buffer as "ReadyToRead" on demand and accessible via "pDataToRead"  (e.g. if no more data need to be recorded)
{attribute 'enable_dynamic_creation'}
FUNCTION_BLOCK DoubleBuffer
VAR_OUTPUT CONSTANT 	
END_VAR                     								
VAR_INPUT
	Overwrite												:	BOOL ; //Overwrite buffer read buffer if not released -> setReadyToRead(FALSE)        
	SizeOfMemory											: 	UDINT := 5120;	//Total size of dynamic allocated buffer (will be splited in half)	   								
END_VAR                     								
VAR_IN_OUT                  								
END_VAR                     								
VAR_OUTPUT       
	TimeFillBuffer											: 	TIME; //Last elapsed time to fill the buffer and set ReadyToRead=TRUE
	MinTimeFillBuffer										:	TIME; //Min time to fill buffer
	MaxTimeFillBuffer										:	TIME; //Max time to fill buffer
	Full													:	BOOL; //Buffer is full
	Empty													:	BOOL := TRUE; //Buffer is empty 
	ReadyToRead												:	BOOL; //TRUE = Data are ready and can be read via "pDataToRead" to process 
	pDataToRead												:	POINTER TO BYTE; //Pointer to recorded data/filled buffer	
	SizeOfDataToRead										:	UDINT; //Count of bytes in filled buffer ready to ready 
{attribute 'displaymode':='hex'}
	hr														:	HRESULT; //Last result of method call
END_VAR                     								
VAR            
//local ************************************************************************************
	Interlock												:	BOOL; //Task interlock
	Buffer2Active											:	BOOL; //Indicates active buffer pointer 
	pBuffer1												: 	POINTER TO BYTE; //Pointer to start of allocated memory
	pBuffer2												: 	POINTER TO BYTE; //Pointer to second half of allocated memory
	StartTimeFillBuffer										:	TIME;
	
	MemSizeOfAllocatedMemory								: 	UDINT; //Total size of allocated memory
	MemSizeOfBuffer											: 	UDINT; //Size of split buffer
	MemSizeOfWriteBuffer									:	UDINT; //Actual size of recorded data


//trigger *********************************************************************************

//timer ***********************************************************************************

//instances ***********************************************************************************             								

//Dummys ****************************************************************************************

END_VAR

METHOD PUBLIC addData : HRESULT //Add data to write buffer and sets "ReadyToRead" if buffer is filled and data can be read to process 
VAR_INPUT
	pData													:	POINTER TO BYTE;
	SizeofData												:	UDINT;
END_VAR

IF pData <> 0 
THEN		
	//Allocate Memory to buffer messages
	IF pBuffer1 = 0
		OR SizeOfMemory > MemSizeOfAllocatedMemory 
	THEN //Allocate full memory with first entry 		
		IF NOT Allocate(SizeOfMemory)
		THEN
			addData := hr										:= E_HRESULTADSERR.NOMEMORY;
			RETURN;														
		END_IF					
	END_IF	

	IF MemSizeOfWriteBuffer = 0 THEN StartTimeFillBuffer := TIME(); END_IF
	
	//Change buffer if filled
	IF SizeofData + MemSizeOfWriteBuffer >= MemSizeOfBuffer
	THEN
		IF setReadyToRead(TRUE) <> S_OK
		THEN
			addData 											:= hr;
			RETURN;
		END_IF
	ELSE
		Full													:= FALSE;
		Empty													:= FALSE;
	END_IF
			
	//Copy data to buffer
	MEMCPY(SEL(Buffer2Active, pBuffer1, pBuffer2) + MemSizeOfWriteBuffer, pData, SizeofData);
	MemSizeOfWriteBuffer										:= MemSizeOfWriteBuffer + SizeofData;
	
	addData := hr												:= S_OK;
ELSE
	addData := hr												:= E_HRESULTADSERR.INVALIDPARM;
END_IF
END_METHOD

METHOD PUBLIC addString : HRESULT //Add string to write buffer and sets "ReadyToRead" if buffer is filled and data can be read to process 
VAR_INPUT
	Data													:	T_MAXSTRING;
END_VAR
addString := hr := addData(ADR(Data),TO_UDINT(LEN(Data)));
END_METHOD

METHOD PROTECTED FINAL allocate : BOOL //allocte buffer memory form router pool
VAR_INPUT
	SizeOfBuffer											:	UDINT;
END_VAR
VAR
	pDummy													:	POINTER TO BYTE;	
End_Var
IF SizeOfBuffer	= 0
THEN
	Allocate												:= FALSE;
	
ELSIF pBuffer1 = 0
THEN
	MemSizeOfAllocatedMemory								:= SizeOfBuffer;
	pBuffer1												:= __NEW(BYTE,MemSizeOfAllocatedMemory );
	MemSizeOfBuffer											:= MemSizeOfAllocatedMemory / 2;
	pBuffer2												:= pBuffer1 + MemSizeOfBuffer; 
	Buffer2Active											:= FALSE;
	MemSizeOfWriteBuffer									:= 0;
	
	IF PARAM.ENABLE_DEBUG_MSG_DYNAMIC_MEM_ALLOCATION
	THEN
		AdsLogHint('EngineeringToolbox | FB DoubleBuffer | An instance allocated %s bytes from the dynamic memory of the ADS router memory pool', TO_STRING(MemSizeOfAllocatedMemory));
	END_IF	
	Allocate												:= TRUE;
ELSIF SizeOfBuffer > MemSizeOfBuffer 
THEN //Since increased, allocate new memory
	
	pDummy													:= __NEW(BYTE, SizeOfBuffer); 

	IF SizeOfBuffer > MemSizeOfAllocatedMemory
	THEN //Size increased rescue data from old memory
		IF Buffer2Active
		THEN
			MEMCPY(pDummy,pBuffer2, MemSizeOfBuffer);
		ELSE
			MEMCPY(pDummy,pBuffer1, MemSizeOfBuffer);	
		END_IF
	END_IF

	__DELETE(pBuffer1);  //Delete reference to old memory
	
	MemSizeOfAllocatedMemory								:= SizeOfBuffer;
	pBuffer1												:= pDummy; //Take over new pointer to new memory
	Buffer2Active											:= FALSE;
	MemSizeOfBuffer											:= MemSizeOfAllocatedMemory / 2;
	pBuffer2												:= pBuffer1 + MemSizeOfBuffer; 
	MemSizeOfWriteBuffer										:= 0;
	
	IF PARAM.ENABLE_DEBUG_MSG_DYNAMIC_MEM_ALLOCATION
	THEN
		AdsLogWarn('EngineeringToolbox | FB DoubleBuffer | Value of "SizeOfMemory" increased and an instance has an additional %s bytes allocated from the dynamic memory of the ADS router memory pool', TO_STRING(MemSizeOfAllocatedMemory));
	END_IF
	
	Allocate												:= TRUE;
	
ELSE //Size decreased
	Allocate												:= TRUE;
END_IF
END_METHOD

METHOD PUBLIC copyData : HRESULT //Copy data from buffer (pDataToRead) into destination and reset "ReadyToReady" back to false if succeful executed 
VAR_INPUT
	pDest													:	POINTER TO BYTE; 
	SizeOfDest												:	UDINT; //Size of destination/data to copy
END_VAR
IF pDest <> 0 AND SizeOfDest > 0
	AND pDataToRead <> 0 
THEN
	MEMCPY(pDest, pDataToRead, MIN(SizeOfDest,SizeOfDataToRead));										
	hr		 												:= setReadyToRead(FALSE);	
	
ELSE
	IF pDataToRead = 0
	THEN
		hr													:= E_HRESULTADSERR.NOTREADY;
	ELSIF pDest = 0 
	THEN 
		hr													:= E_HRESULTADSERR.INVALIDPARM;
	ELSIF SizeOfDest = 0
	THEN
		hr													:= E_HRESULTADSERR.INVALIDPARM;	
	END_IF
END_IF
copyData													:= hr;
END_METHOD

METHOD FB_exit : BOOL
VAR_INPUT
	bInCopyCode : BOOL; // if TRUE, the exit method is called for exiting an instance that is copied afterwards (online change).
END_VAR
IF NOT bInCopyCode AND pBuffer1 <> 0
THEN //Release memory in case the PLC stopps
	__DELETE(pBuffer1);
END_IF
END_METHOD

{attribute 'monitoring' := 'call'}
PROPERTY PUBLIC fillLevel : INT //Buffer fill level 100% if both parts of buffer are filled
GET
IF MemSizeOfBuffer <> 0
THEN
	fillLevel												:= 	TO_INT((50.0 / TO_LREAL(MemSizeOfBuffer)) * TO_LREAL(MemSizeOfWriteBuffer))
																+ SEL(ReadyToRead, 0, TO_INT((50.0 / TO_LREAL(MemSizeOfBuffer)) * TO_LREAL(SizeOfDataToRead)));
ELSE
	fillLevel												:= 0;
END_IF
END_GET
END_PROPERTY

//Reset buffer 
METHOD PUBLIC reset : BOOL //TRUE if method is finnished
VAR_INPUT
END_VAR
TimeFillBuffer												:= T#0MS;
MinTimeFillBuffer											:= T#0MS;
MaxTimeFillBuffer											:= T#0MS;
Full														:= FALSE; //Buffer is full
Empty														:= TRUE; //Buffer is empty 
ReadyToRead													:= FALSE;
SizeOfDataToRead											:= 0;
hr															:= S_OK;
MemSizeOfWriteBuffer										:= 0;
reset														:= TRUE;
END_METHOD

METHOD PUBLIC setReadyToRead : HRESULT //Status = FALSE to reset "ReadyToRead" and unlock buffer / Status = TRUE to mark current write buffer as filled and "ReadyToRead", accessible via "pDataToRead"
VAR_INPUT
	Status								:	BOOL; //FALSE to reset "ReadyToRead" or TRUE to set "ReadyToRead" and swap buffer 
END_VAR
IF TestAndSet(Interlock)
THEN
	IF NOT Status
	THEN
		ReadyToRead									:= FALSE;
		Full										:= FALSE;
		Empty										:= MemSizeOfWriteBuffer = 0;
		hr											:= S_OK;
	ELSIF Overwrite 
		OR NOT ReadyToRead
	THEN //Set ready to ready and swap buffer
		hr											:= SEL(swapBuffer(), E_HRESULTADSERR.ABORTED ,S_OK);
		TimeFillBuffer								:= TIME() - StartTimeFillBuffer;
		IF MinTimeFillBuffer = T#0MS THEN MinTimeFillBuffer := TimeFillBuffer; ELSE MinTimeFillBuffer := MIN(TimeFillBuffer,MinTimeFillBuffer); END_IF	
		MaxTimeFillBuffer							:= MAX(TimeFillBuffer,MaxTimeFillBuffer);
		StartTimeFillBuffer							:= TIME();
		ReadyToRead									:= SizeOfDataToRead > 0;
		Full										:= FALSE;
		Empty										:= NOT ReadyToRead;
	ELSE
		TimeFillBuffer								:= TIME() - StartTimeFillBuffer;
		IF MinTimeFillBuffer = T#0MS THEN MinTimeFillBuffer := TimeFillBuffer; ELSE MinTimeFillBuffer := MIN(TimeFillBuffer,MinTimeFillBuffer); END_IF
		MaxTimeFillBuffer							:= MAX(TimeFillBuffer,MaxTimeFillBuffer);
		StartTimeFillBuffer							:= TIME();		
		Full										:= TRUE;
		Empty										:= FALSE;
		hr											:= E_HRESULTADSERR.ABORTED;	
	END_IF
		
	setReadyToRead									:= hr;
	Interlock										:= FALSE;
ELSE
	setReadyToRead									:= E_HRESULTADSERR.BUSY;
END_IF
END_METHOD

METHOD PROTECTED FINAL swapBuffer : BOOL //swap write and read buffer and asign filled buffer to pDataToRead
VAR_INPUT
END_VAR
pDataToRead													:= SEL(Buffer2Active, pBuffer1, pBuffer2);
SizeOfDataToRead											:= MemSizeOfWriteBuffer;	

Buffer2Active												:= NOT Buffer2Active;	

MemSizeOfWriteBuffer										:= 0;
swapBuffer													:= TRUE;
END_METHOD

END_FUNCTION_BLOCK

// POUs/DataBuffer/Quicksort
// this funktionblock sorts an array of struct by an contained element with quicksort routine
// Udpate: compare with static PivotElement
// Find Explanation under https://www.youtube.com/watch?v=eNUM23f6g-s&ab_channel=Studyflix
{attribute 'enable_dynamic_creation'}
FUNCTION_BLOCK Quicksort
VAR CONSTANT
	MAX_STRING_LENGTH										:	INT := PARAM.QUICKSORT_MAX_STRING_LENGTH;
	MAX_WSTRING_LENGTH										:	INT := PARAM.QUICKSORT_MAX_WSTRING_LENGTH;
END_VAR
VAR_INPUT
	SortInverse												:	BOOL := FALSE;//inverses order of content
	IgnoreBlank												:	BOOL := FALSE;//sort blank characters at last			
END_VAR
VAR_OUTPUT
END_VAR
VAR
	pElement_Tmp											:	POINTER TO BYTE;		// Copy Pointer 3 - allocated memory
	MemSizeOfStruct											:	UDINT;
END_VAR

;

